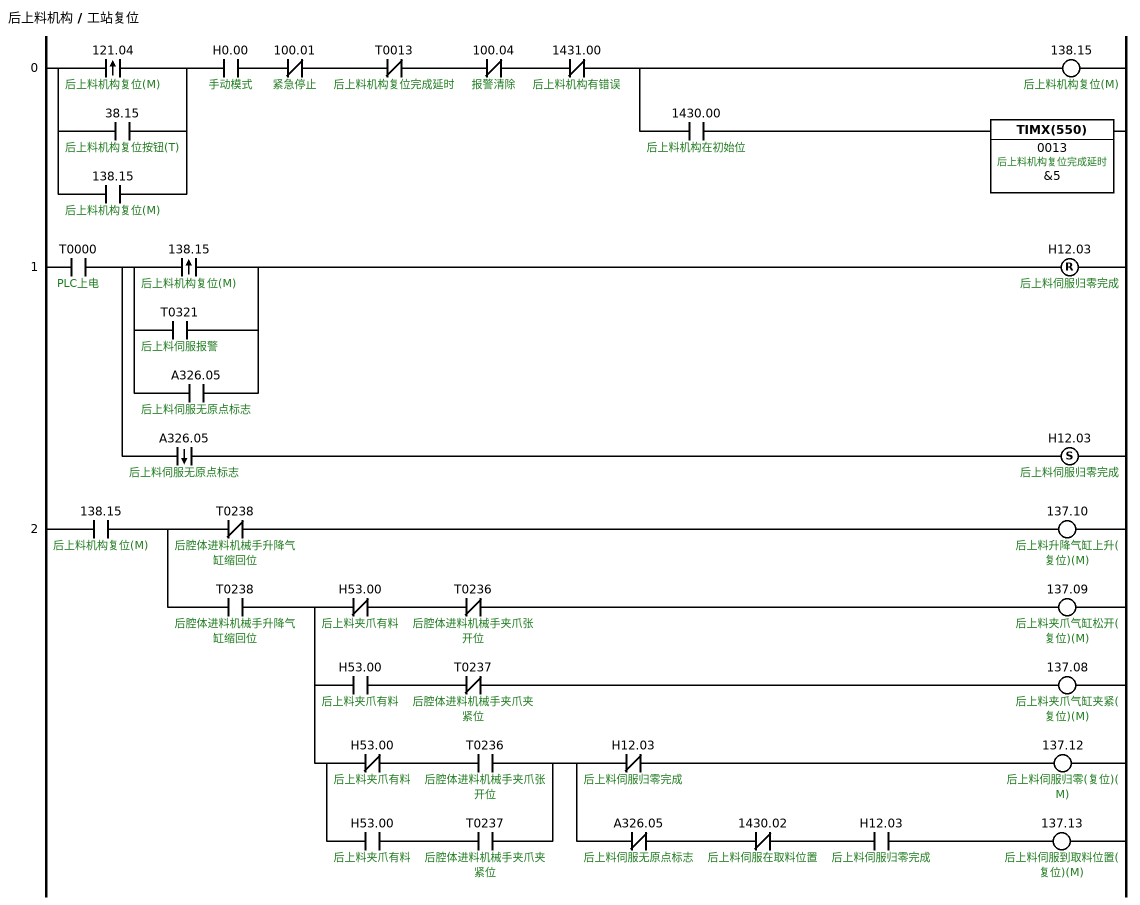
; rung 0
@LD 121.04  ; 后上料机构复位(M)
OR 38.15  ; 后上料机构复位按钮(T)
OR 138.15  ; 后上料机构复位(M)
AND H0.00  ; 手动模式
ANDNOT 100.01  ; 紧急停止
ANDNOT T0013  ; 后上料机构复位完成延时
ANDNOT 100.04  ; 报警清除
ANDNOT 1431.00  ; 后上料机构有错误
OUT 138.15  ; 后上料机构复位(M)
AND 1430.00  ; 后上料机构在初始位
TIMX(550) 0013 &5  ; 后上料机构复位完成延时
; rung 1
LD T0000  ; PLC上电
OUT TR0
@LD 138.15  ; 后上料机构复位(M)
OR T0321  ; 后上料伺服报警
OR A326.05  ; 后上料伺服无原点标志
ANDLD
RSET H12.03  ; 后上料伺服归零完成
LD TR0
%AND A326.05  ; 后上料伺服无原点标志
SET H12.03  ; 后上料伺服归零完成
; rung 2
LD 138.15  ; 后上料机构复位(M)
OUT TR0
ANDNOT T0238  ; 后腔体进料机械手升降气缸缩回位
OUT 137.10  ; 后上料升降气缸上升(复位)(M)
LD TR0
AND T0238  ; 后腔体进料机械手升降气缸缩回位
OUT TR0
ANDNOT H53.00  ; 后上料夹爪有料
ANDNOT T0236  ; 后腔体进料机械手夹爪张开位
OUT 137.09  ; 后上料夹爪气缸松开(复位)(M)
LD TR0
AND H53.00  ; 后上料夹爪有料
ANDNOT T0237  ; 后腔体进料机械手夹爪夹紧位
OUT 137.08  ; 后上料夹爪气缸夹紧(复位)(M)
LD TR0
LDNOT H53.00  ; 后上料夹爪有料
AND T0236  ; 后腔体进料机械手夹爪张开位
LD H53.00  ; 后上料夹爪有料
AND T0237  ; 后腔体进料机械手夹爪夹紧位
ORLD
ANDLD
OUT TR0
ANDNOT H12.03  ; 后上料伺服归零完成
OUT 137.12  ; 后上料伺服归零(复位)(M)
LD TR0
ANDNOT A326.05  ; 后上料伺服无原点标志
ANDNOT 1430.02  ; 后上料伺服在取料位置
AND H12.03  ; 后上料伺服归零完成
OUT 137.13  ; 后上料伺服到取料位置(复位)(M)

### Section 手动操作

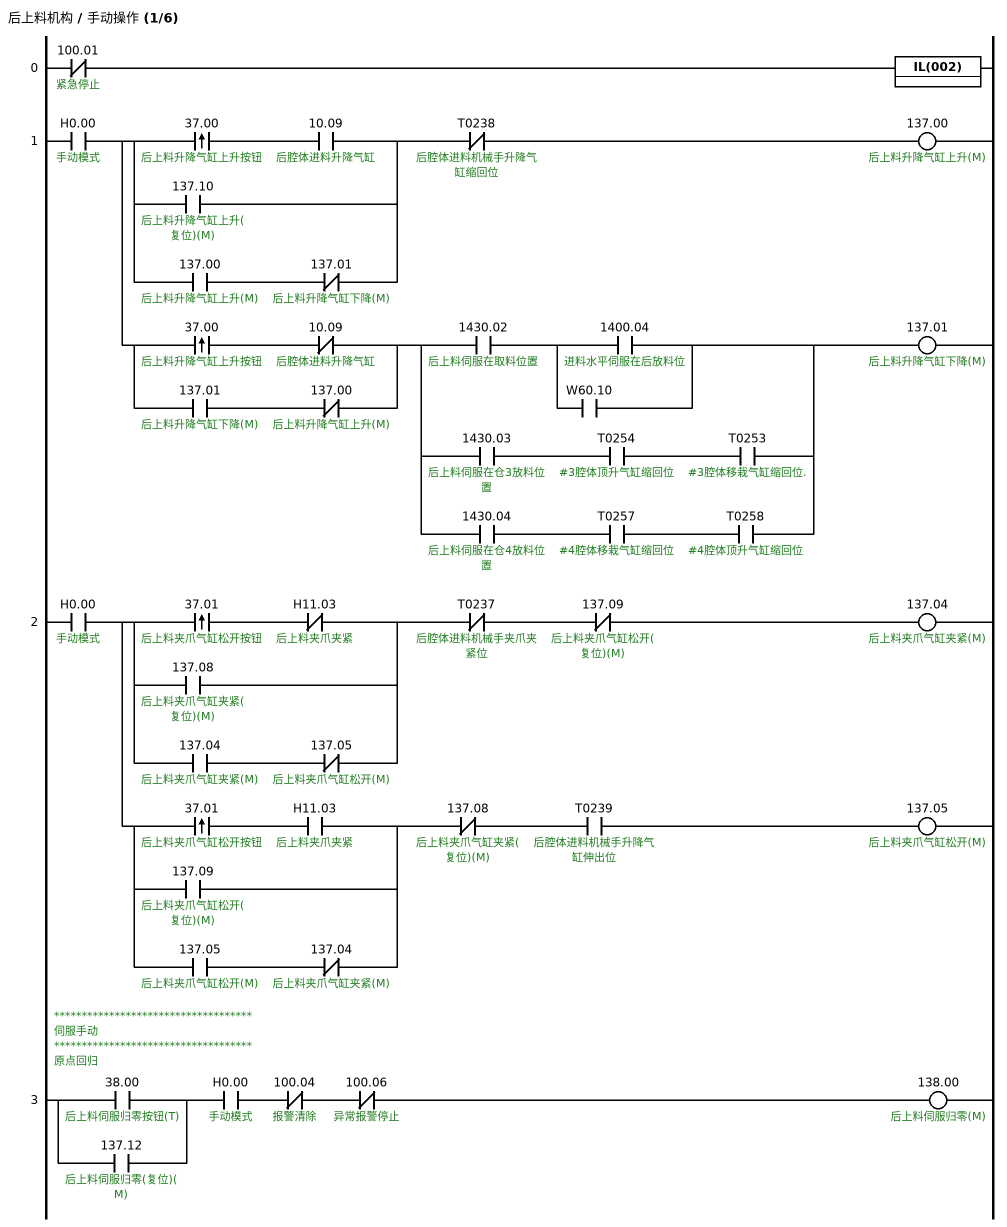
; rung 0
LDNOT 100.01  ; 紧急停止
IL(002)
; rung 1
LD H0.00  ; 手动模式
OUT TR0
@LD 37.00  ; 后上料升降气缸上升按钮
AND 10.09  ; 后腔体进料升降气缸
OR 137.10  ; 后上料升降气缸上升(复位)(M)
LD 137.00  ; 后上料升降气缸上升(M)
ANDNOT 137.01  ; 后上料升降气缸下降(M)
ORLD
ANDLD
ANDNOT T0238  ; 后腔体进料机械手升降气缸缩回位
OUT 137.00  ; 后上料升降气缸上升(M)
LD TR0
@LD 37.00  ; 后上料升降气缸上升按钮
ANDNOT 10.09  ; 后腔体进料升降气缸
LD 137.01  ; 后上料升降气缸下降(M)
ANDNOT 137.00  ; 后上料升降气缸上升(M)
ORLD
ANDLD
LD 1430.02  ; 后上料伺服在取料位置
LD 1400.04  ; 进料水平伺服在后放料位
OR W60.10
ANDLD
LD 1430.03  ; 后上料伺服在仓3放料位置
AND T0254  ; #3腔体顶升气缸缩回位
AND T0253  ; #3腔体移栽气缸缩回位.
ORLD
LD 1430.04  ; 后上料伺服在仓4放料位置
AND T0257  ; #4腔体移栽气缸缩回位
AND T0258  ; #4腔体顶升气缸缩回位
ORLD
ANDLD
OUT 137.01  ; 后上料升降气缸下降(M)
; rung 2
LD H0.00  ; 手动模式
OUT TR0
@LD 37.01  ; 后上料夹爪气缸松开按钮
ANDNOT H11.03  ; 后上料夹爪夹紧
OR 137.08  ; 后上料夹爪气缸夹紧(复位)(M)
LD 137.04  ; 后上料夹爪气缸夹紧(M)
ANDNOT 137.05  ; 后上料夹爪气缸松开(M)
ORLD
ANDLD
ANDNOT T0237  ; 后腔体进料机械手夹爪夹紧位
ANDNOT 137.09  ; 后上料夹爪气缸松开(复位)(M)
OUT 137.04  ; 后上料夹爪气缸夹紧(M)
LD TR0
@LD 37.01  ; 后上料夹爪气缸松开按钮
AND H11.03  ; 后上料夹爪夹紧
OR 137.09  ; 后上料夹爪气缸松开(复位)(M)
LD 137.05  ; 后上料夹爪气缸松开(M)
ANDNOT 137.04  ; 后上料夹爪气缸夹紧(M)
ORLD
ANDLD
ANDNOT 137.08  ; 后上料夹爪气缸夹紧(复位)(M)
AND T0239  ; 后腔体进料机械手升降气缸伸出位
OUT 137.05  ; 后上料夹爪气缸松开(M)
; rung 3: ************************************ / 伺服手动 / ************************************ / 原点回归
LD 38.00  ; 后上料伺服归零按钮(T)
OR 137.12  ; 后上料伺服归零(复位)(M)
AND H0.00  ; 手动模式
ANDNOT 100.04  ; 报警清除
ANDNOT 100.06  ; 异常报警停止
OUT 138.00  ; 后上料伺服归零(M)

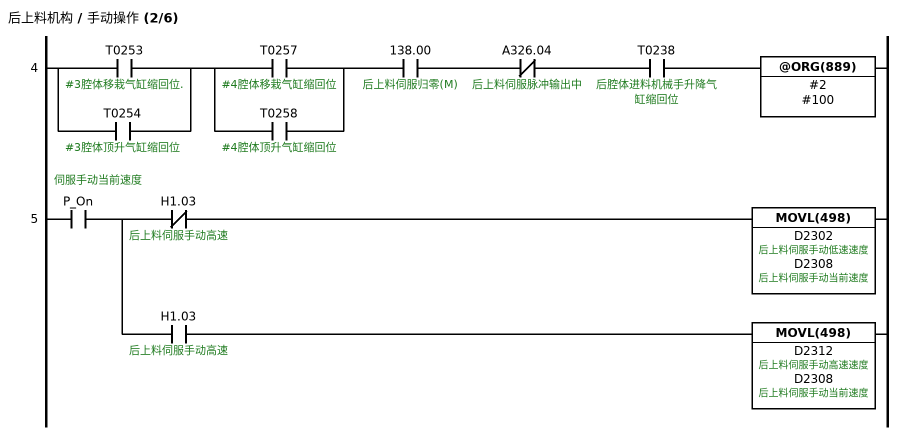
; rung 4
LD T0253  ; #3腔体移栽气缸缩回位.
OR T0254  ; #3腔体顶升气缸缩回位
LD T0257  ; #4腔体移栽气缸缩回位
OR T0258  ; #4腔体顶升气缸缩回位
ANDLD
AND 138.00  ; 后上料伺服归零(M)
ANDNOT A326.04  ; 后上料伺服脉冲输出中
AND T0238  ; 后腔体进料机械手升降气缸缩回位
@ORG(889) #2 #100
; rung 5: 伺服手动当前速度
LD P_On
OUT TR0
ANDNOT H1.03  ; 后上料伺服手动高速
MOVL(498) D2302 D2308  ; 后上料伺服手动低速速度, 后上料伺服手动当前速度
LD TR0
AND H1.03  ; 后上料伺服手动高速
MOVL(498) D2312 D2308  ; 后上料伺服手动高速速度, 后上料伺服手动当前速度

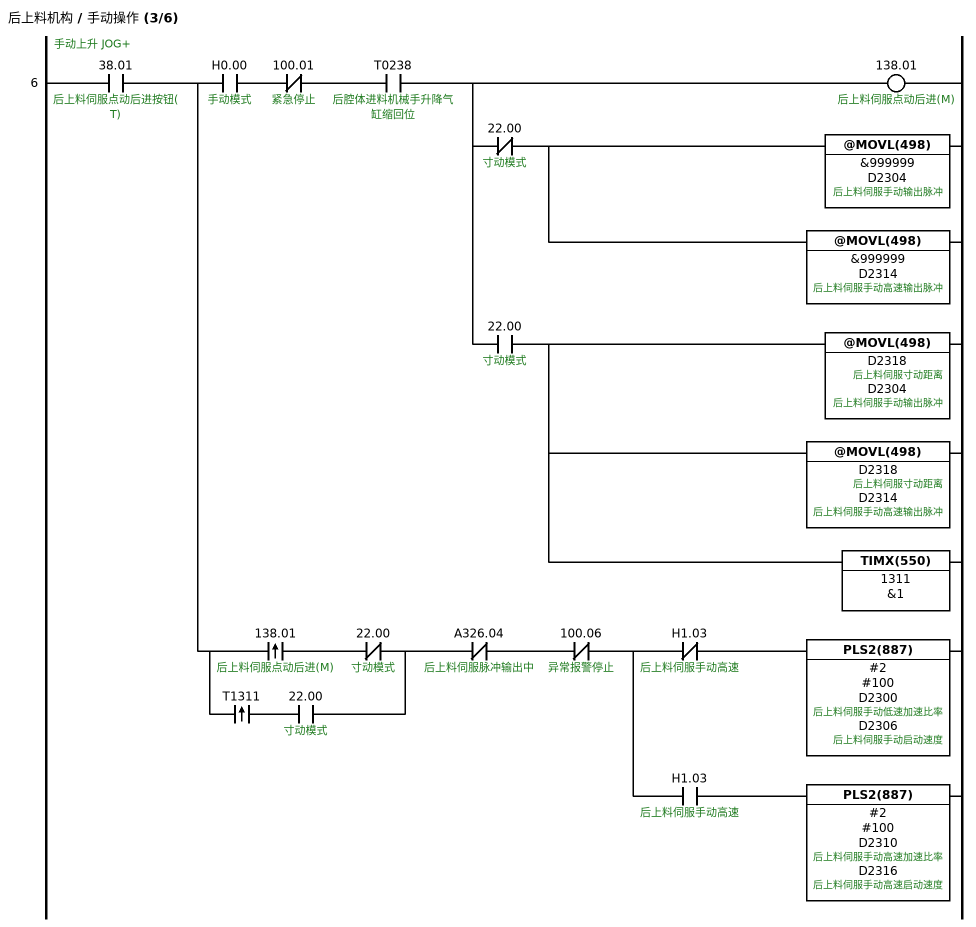
; rung 6: 手动上升 JOG+
LD 38.01  ; 后上料伺服点动后进按钮(T)
OUT TR0
AND H0.00  ; 手动模式
ANDNOT 100.01  ; 紧急停止
AND T0238  ; 后腔体进料机械手升降气缸缩回位
OUT TR1
OUT 138.01  ; 后上料伺服点动后进(M)
ANDNOT 22.00  ; 寸动模式
@MOVL(498) &999999 D2304  ; 后上料伺服手动输出脉冲
@MOVL(498) &999999 D2314  ; 后上料伺服手动高速输出脉冲
LD TR1
AND 22.00  ; 寸动模式
@MOVL(498) D2318 D2304  ; 后上料伺服寸动距离, 后上料伺服手动输出脉冲
@MOVL(498) D2318 D2314  ; 后上料伺服寸动距离, 后上料伺服手动高速输出脉冲
TIMX(550) 1311 &1
LD TR0
@LD 138.01  ; 后上料伺服点动后进(M)
ANDNOT 22.00  ; 寸动模式
@LD T1311
AND 22.00  ; 寸动模式
ORLD
ANDLD
ANDNOT A326.04  ; 后上料伺服脉冲输出中
ANDNOT 100.06  ; 异常报警停止
OUT TR0
ANDNOT H1.03  ; 后上料伺服手动高速
PLS2(887) #2 #100 D2300 D2306  ; 后上料伺服手动低速加速比率, 后上料伺服手动启动速度
LD TR0
AND H1.03  ; 后上料伺服手动高速
PLS2(887) #2 #100 D2310 D2316  ; 后上料伺服手动高速加速比率, 后上料伺服手动高速启动速度

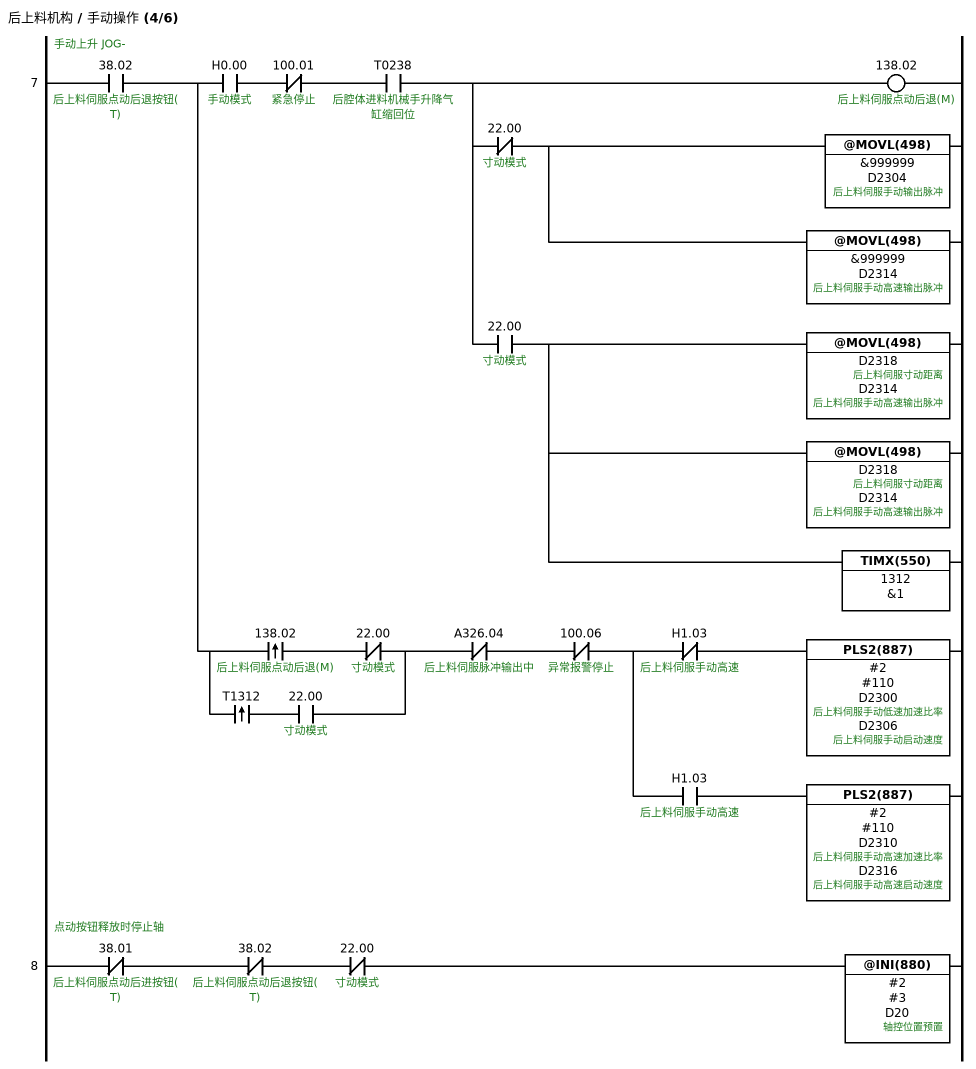
; rung 7: 手动上升 JOG-
LD 38.02  ; 后上料伺服点动后退按钮(T)
OUT TR0
AND H0.00  ; 手动模式
ANDNOT 100.01  ; 紧急停止
AND T0238  ; 后腔体进料机械手升降气缸缩回位
OUT TR1
OUT 138.02  ; 后上料伺服点动后退(M)
ANDNOT 22.00  ; 寸动模式
@MOVL(498) &999999 D2304  ; 后上料伺服手动输出脉冲
@MOVL(498) &999999 D2314  ; 后上料伺服手动高速输出脉冲
LD TR1
AND 22.00  ; 寸动模式
@MOVL(498) D2318 D2314  ; 后上料伺服寸动距离, 后上料伺服手动高速输出脉冲
@MOVL(498) D2318 D2314  ; 后上料伺服寸动距离, 后上料伺服手动高速输出脉冲
TIMX(550) 1312 &1
LD TR0
@LD 138.02  ; 后上料伺服点动后退(M)
ANDNOT 22.00  ; 寸动模式
@LD T1312
AND 22.00  ; 寸动模式
ORLD
ANDLD
ANDNOT A326.04  ; 后上料伺服脉冲输出中
ANDNOT 100.06  ; 异常报警停止
OUT TR0
ANDNOT H1.03  ; 后上料伺服手动高速
PLS2(887) #2 #110 D2300 D2306  ; 后上料伺服手动低速加速比率, 后上料伺服手动启动速度
LD TR0
AND H1.03  ; 后上料伺服手动高速
PLS2(887) #2 #110 D2310 D2316  ; 后上料伺服手动高速加速比率, 后上料伺服手动高速启动速度
; rung 8: 点动按钮释放时停止轴
LDNOT 38.01  ; 后上料伺服点动后进按钮(T)
ANDNOT 38.02  ; 后上料伺服点动后退按钮(T)
ANDNOT 22.00  ; 寸动模式
@INI(880) #2 #3 D20  ; 轴控位置预置

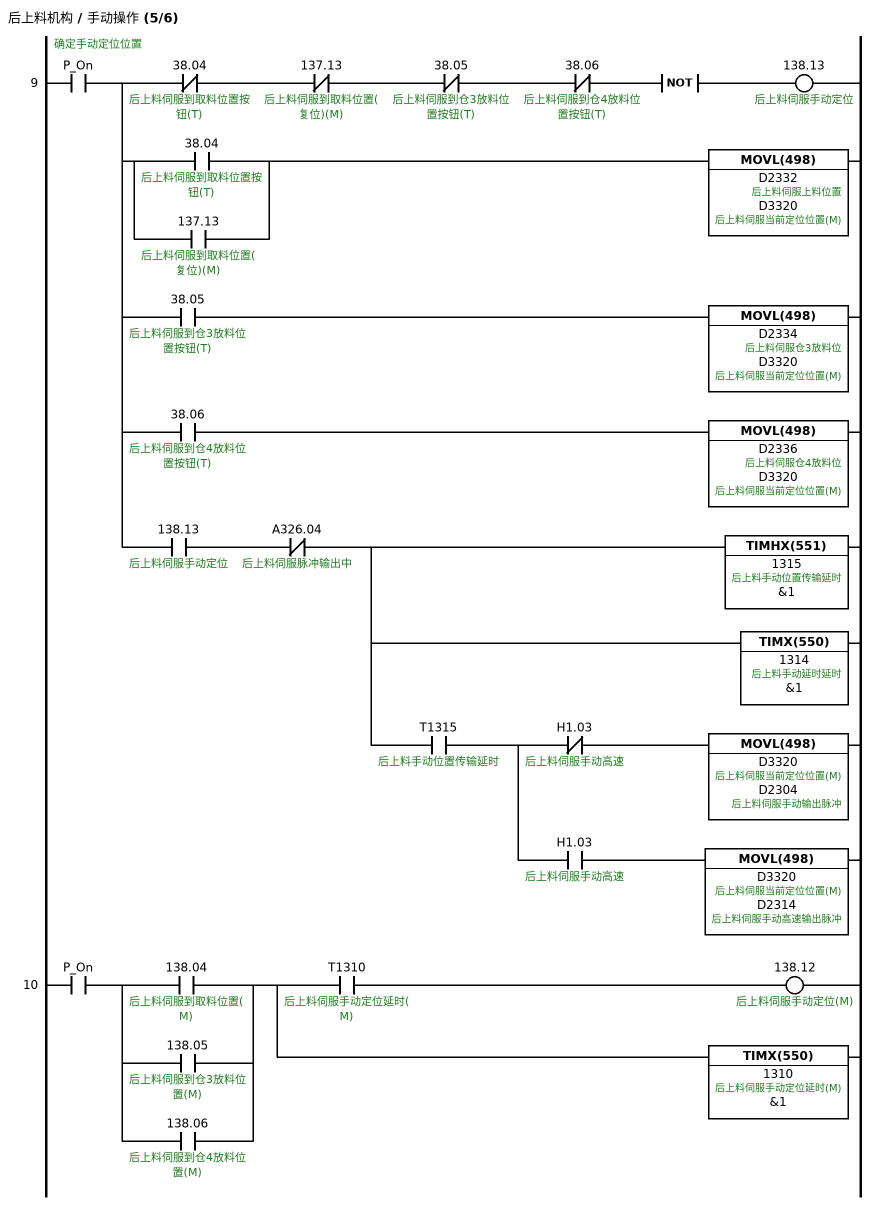
; rung 9: 确定手动定位位置
LD P_On
OUT TR0
ANDNOT 38.04  ; 后上料伺服到取料位置按钮(T)
ANDNOT 137.13  ; 后上料伺服到取料位置(复位)(M)
ANDNOT 38.05  ; 后上料伺服到仓3放料位置按钮(T)
ANDNOT 38.06  ; 后上料伺服到仓4放料位置按钮(T)
NOT(520)
OUT 138.13  ; 后上料伺服手动定位
LD TR0
LD 38.04  ; 后上料伺服到取料位置按钮(T)
OR 137.13  ; 后上料伺服到取料位置(复位)(M)
ANDLD
MOVL(498) D2332 D3320  ; 后上料伺服上料位置, 后上料伺服当前定位位置(M)
LD TR0
AND 38.05  ; 后上料伺服到仓3放料位置按钮(T)
MOVL(498) D2334 D3320  ; 后上料伺服仓3放料位, 后上料伺服当前定位位置(M)
LD TR0
AND 38.06  ; 后上料伺服到仓4放料位置按钮(T)
MOVL(498) D2336 D3320  ; 后上料伺服仓4放料位, 后上料伺服当前定位位置(M)
LD TR0
AND 138.13  ; 后上料伺服手动定位
ANDNOT A326.04  ; 后上料伺服脉冲输出中
TIMHX(551) 1315 &1  ; 后上料手动位置传输延时
TIMX(550) 1314 &1  ; 后上料手动延时延时
AND T1315  ; 后上料手动位置传输延时
OUT TR0
ANDNOT H1.03  ; 后上料伺服手动高速
MOVL(498) D3320 D2304  ; 后上料伺服当前定位位置(M), 后上料伺服手动输出脉冲
LD TR0
AND H1.03  ; 后上料伺服手动高速
MOVL(498) D3320 D2314  ; 后上料伺服当前定位位置(M), 后上料伺服手动高速输出脉冲
; rung 10
LD P_On
LD 138.04  ; 后上料伺服到取料位置(M)
OR 138.05  ; 后上料伺服到仓3放料位置(M)
OR 138.06  ; 后上料伺服到仓4放料位置(M)
ANDLD
OUT TR0
AND T1310  ; 后上料伺服手动定位延时(M)
OUT 138.12  ; 后上料伺服手动定位(M)
LD TR0
TIMX(550) 1310 &1  ; 后上料伺服手动定位延时(M)

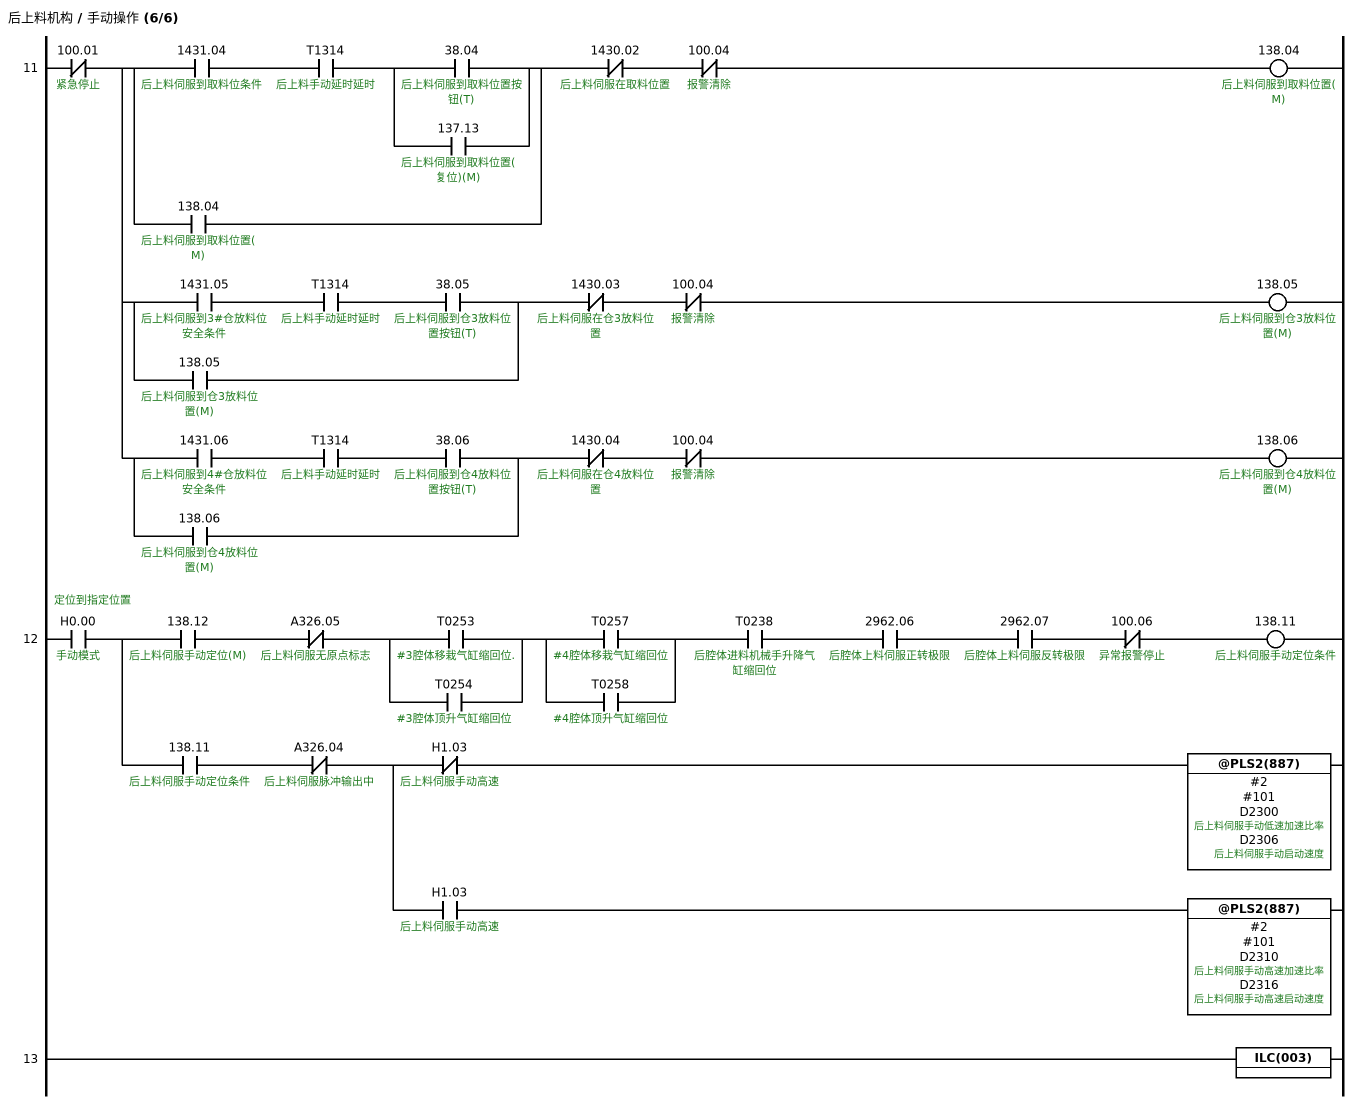
; rung 11
LDNOT 100.01  ; 紧急停止
OUT TR0
LD 1431.04  ; 后上料伺服到取料位条件
AND T1314  ; 后上料手动延时延时
LD 38.04  ; 后上料伺服到取料位置按钮(T)
OR 137.13  ; 后上料伺服到取料位置(复位)(M)
ANDLD
OR 138.04  ; 后上料伺服到取料位置(M)
ANDLD
ANDNOT 1430.02  ; 后上料伺服在取料位置
ANDNOT 100.04  ; 报警清除
OUT 138.04  ; 后上料伺服到取料位置(M)
LD TR0
LD 1431.05  ; 后上料伺服到3#仓放料位安全条件
AND T1314  ; 后上料手动延时延时
AND 38.05  ; 后上料伺服到仓3放料位置按钮(T)
OR 138.05  ; 后上料伺服到仓3放料位置(M)
ANDLD
ANDNOT 1430.03  ; 后上料伺服在仓3放料位置
ANDNOT 100.04  ; 报警清除
OUT 138.05  ; 后上料伺服到仓3放料位置(M)
LD TR0
LD 1431.06  ; 后上料伺服到4#仓放料位安全条件
AND T1314  ; 后上料手动延时延时
AND 38.06  ; 后上料伺服到仓4放料位置按钮(T)
OR 138.06  ; 后上料伺服到仓4放料位置(M)
ANDLD
ANDNOT 1430.04  ; 后上料伺服在仓4放料位置
ANDNOT 100.04  ; 报警清除
OUT 138.06  ; 后上料伺服到仓4放料位置(M)
; rung 12: 定位到指定位置
LD H0.00  ; 手动模式
OUT TR0
AND 138.12  ; 后上料伺服手动定位(M)
ANDNOT A326.05  ; 后上料伺服无原点标志
LD T0253  ; #3腔体移栽气缸缩回位.
OR T0254  ; #3腔体顶升气缸缩回位
ANDLD
LD T0257  ; #4腔体移栽气缸缩回位
OR T0258  ; #4腔体顶升气缸缩回位
ANDLD
AND T0238  ; 后腔体进料机械手升降气缸缩回位
AND 2962.06  ; 后腔体上料伺服正转极限
AND 2962.07  ; 后腔体上料伺服反转极限
ANDNOT 100.06  ; 异常报警停止
OUT 138.11  ; 后上料伺服手动定位条件
LD TR0
AND 138.11  ; 后上料伺服手动定位条件
ANDNOT A326.04  ; 后上料伺服脉冲输出中
OUT TR0
ANDNOT H1.03  ; 后上料伺服手动高速
@PLS2(887) #2 #101 D2300 D2306  ; 后上料伺服手动低速加速比率, 后上料伺服手动启动速度
LD TR0
AND H1.03  ; 后上料伺服手动高速
@PLS2(887) #2 #101 D2310 D2316  ; 后上料伺服手动高速加速比率, 后上料伺服手动高速启动速度
; rung 13
ILC(003)

### Section 自动运行

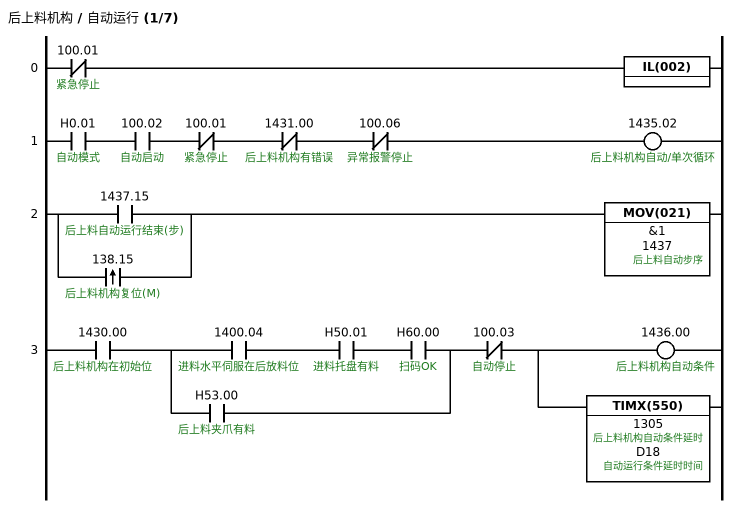
; rung 0
LDNOT 100.01  ; 紧急停止
IL(002)
; rung 1
LD H0.01  ; 自动模式
AND 100.02  ; 自动启动
ANDNOT 100.01  ; 紧急停止
ANDNOT 1431.00  ; 后上料机构有错误
ANDNOT 100.06  ; 异常报警停止
OUT 1435.02  ; 后上料机构自动/单次循环
; rung 2
LD 1437.15  ; 后上料自动运行结束(步)
@OR 138.15  ; 后上料机构复位(M)
MOV(021) &1 1437  ; 后上料自动步序
; rung 3
LD 1430.00  ; 后上料机构在初始位
LD 1400.04  ; 进料水平伺服在后放料位
AND H50.01  ; 进料托盘有料
AND H60.00  ; 扫码OK
OR H53.00  ; 后上料夹爪有料
ANDLD
ANDNOT 100.03  ; 自动停止
OUT 1436.00  ; 后上料机构自动条件
TIMX(550) 1305 D18  ; 自动运行条件延时时间, 后上料机构自动条件延时

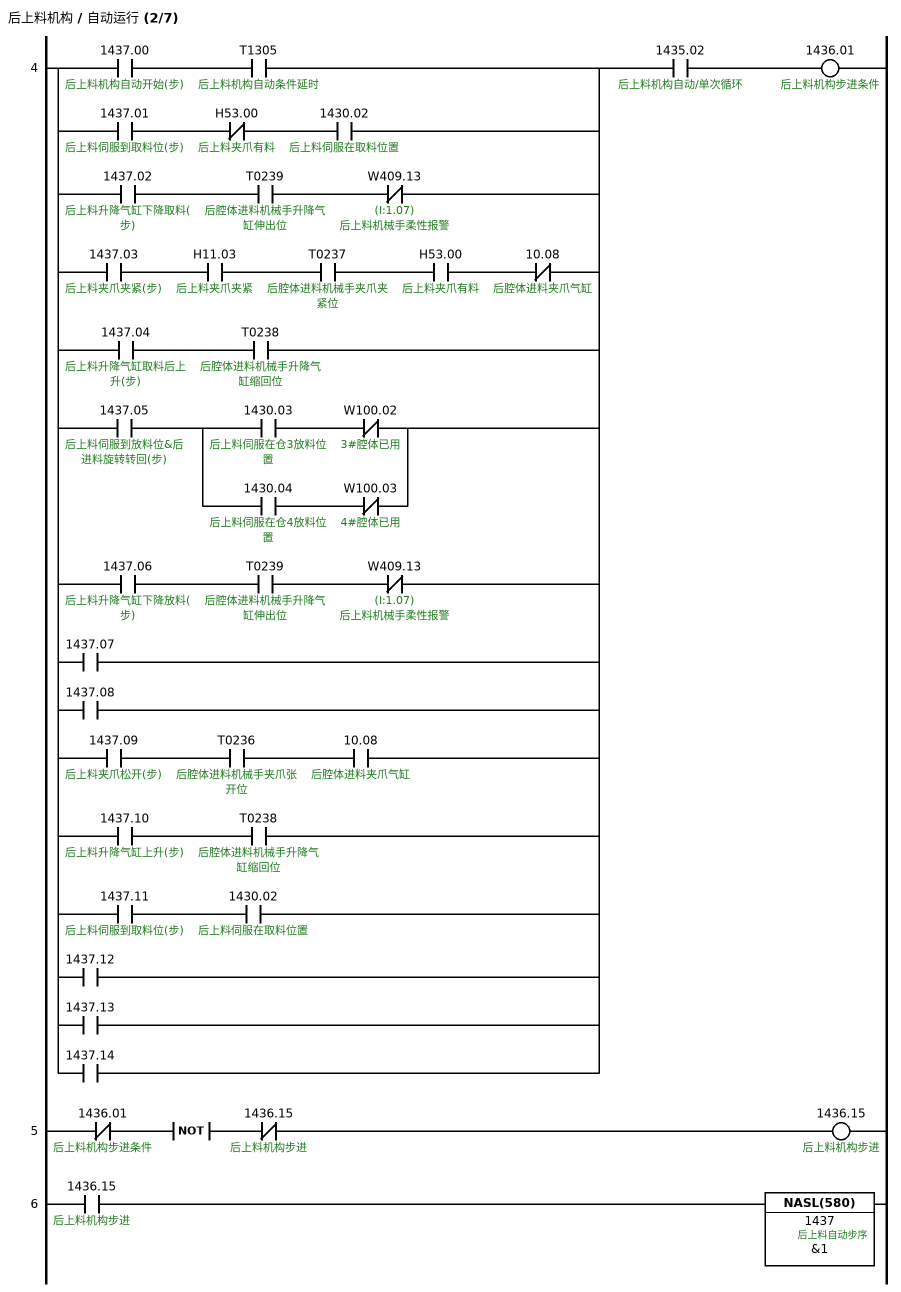
; rung 4
LD 1437.00  ; 后上料机构自动开始(步)
AND T1305  ; 后上料机构自动条件延时
LD 1437.01  ; 后上料伺服到取料位(步)
ANDNOT H53.00  ; 后上料夹爪有料
AND 1430.02  ; 后上料伺服在取料位置
ORLD
LD 1437.02  ; 后上料升降气缸下降取料(步)
AND T0239  ; 后腔体进料机械手升降气缸伸出位
ANDNOT W409.13  ; (I:1.07) 后上料机械手柔性报警
ORLD
LD 1437.03  ; 后上料夹爪夹紧(步)
AND H11.03  ; 后上料夹爪夹紧
AND T0237  ; 后腔体进料机械手夹爪夹紧位
AND H53.00  ; 后上料夹爪有料
ANDNOT 10.08  ; 后腔体进料夹爪气缸
ORLD
LD 1437.04  ; 后上料升降气缸取料后上升(步)
AND T0238  ; 后腔体进料机械手升降气缸缩回位
ORLD
LD 1437.05  ; 后上料伺服到放料位&后进料旋转转回(步)
LD 1430.03  ; 后上料伺服在仓3放料位置
ANDNOT W100.02  ; 3#腔体已用
LD 1430.04  ; 后上料伺服在仓4放料位置
ANDNOT W100.03  ; 4#腔体已用
ORLD
ANDLD
ORLD
LD 1437.06  ; 后上料升降气缸下降放料(步)
AND T0239  ; 后腔体进料机械手升降气缸伸出位
ANDNOT W409.13  ; (I:1.07) 后上料机械手柔性报警
ORLD
OR 1437.07
OR 1437.08
LD 1437.09  ; 后上料夹爪松开(步)
AND T0236  ; 后腔体进料机械手夹爪张开位
AND 10.08  ; 后腔体进料夹爪气缸
ORLD
LD 1437.10  ; 后上料升降气缸上升(步)
AND T0238  ; 后腔体进料机械手升降气缸缩回位
ORLD
LD 1437.11  ; 后上料伺服到取料位(步)
AND 1430.02  ; 后上料伺服在取料位置
ORLD
OR 1437.12
OR 1437.13
OR 1437.14
AND 1435.02  ; 后上料机构自动/单次循环
OUT 1436.01  ; 后上料机构步进条件
; rung 5
LDNOT 1436.01  ; 后上料机构步进条件
NOT(520)
ANDNOT 1436.15  ; 后上料机构步进
OUT 1436.15  ; 后上料机构步进
; rung 6
LD 1436.15  ; 后上料机构步进
NASL(580) 1437 &1  ; 后上料自动步序

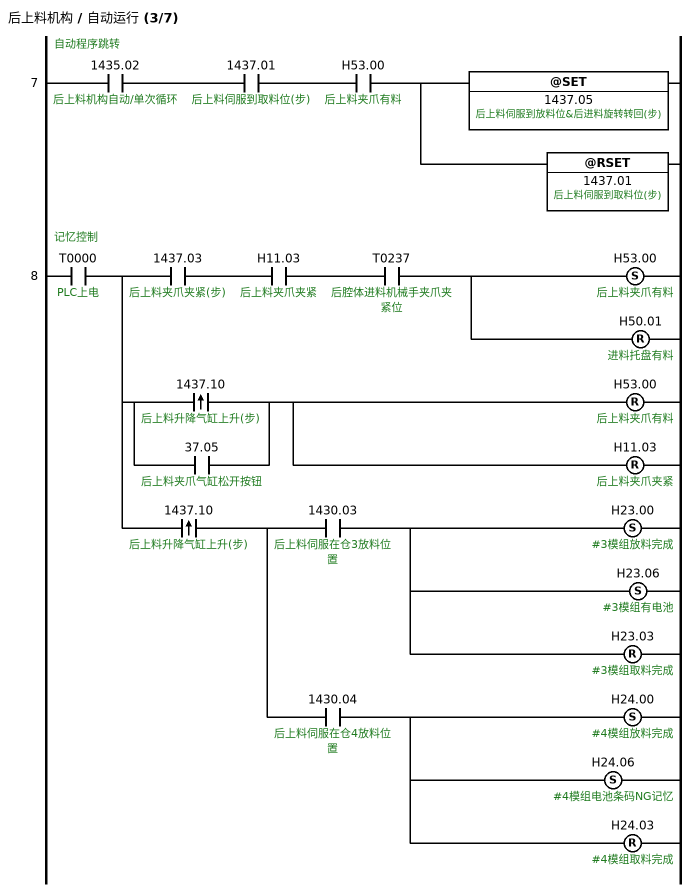
; rung 7: 自动程序跳转
LD 1435.02  ; 后上料机构自动/单次循环
AND 1437.01  ; 后上料伺服到取料位(步)
AND H53.00  ; 后上料夹爪有料
@SET 1437.05  ; 后上料伺服到放料位&后进料旋转转回(步)
@RSET 1437.01  ; 后上料伺服到取料位(步)
; rung 8: 记忆控制
LD T0000  ; PLC上电
OUT TR0
AND 1437.03  ; 后上料夹爪夹紧(步)
AND H11.03  ; 后上料夹爪夹紧
AND T0237  ; 后腔体进料机械手夹爪夹紧位
SET H53.00  ; 后上料夹爪有料
RSET H50.01  ; 进料托盘有料
LD TR0
@LD 1437.10  ; 后上料升降气缸上升(步)
OR 37.05  ; 后上料夹爪气缸松开按钮
ANDLD
RSET H53.00  ; 后上料夹爪有料
RSET H11.03  ; 后上料夹爪夹紧
LD TR0
@AND 1437.10  ; 后上料升降气缸上升(步)
OUT TR0
AND 1430.03  ; 后上料伺服在仓3放料位置
SET H23.00  ; #3模组放料完成
SET H23.06  ; #3模组有电池
RSET H23.03  ; #3模组取料完成
LD TR0
AND 1430.04  ; 后上料伺服在仓4放料位置
SET H24.00  ; #4模组放料完成
SET H24.06  ; #4模组电池条码NG记忆
RSET H24.03  ; #4模组取料完成

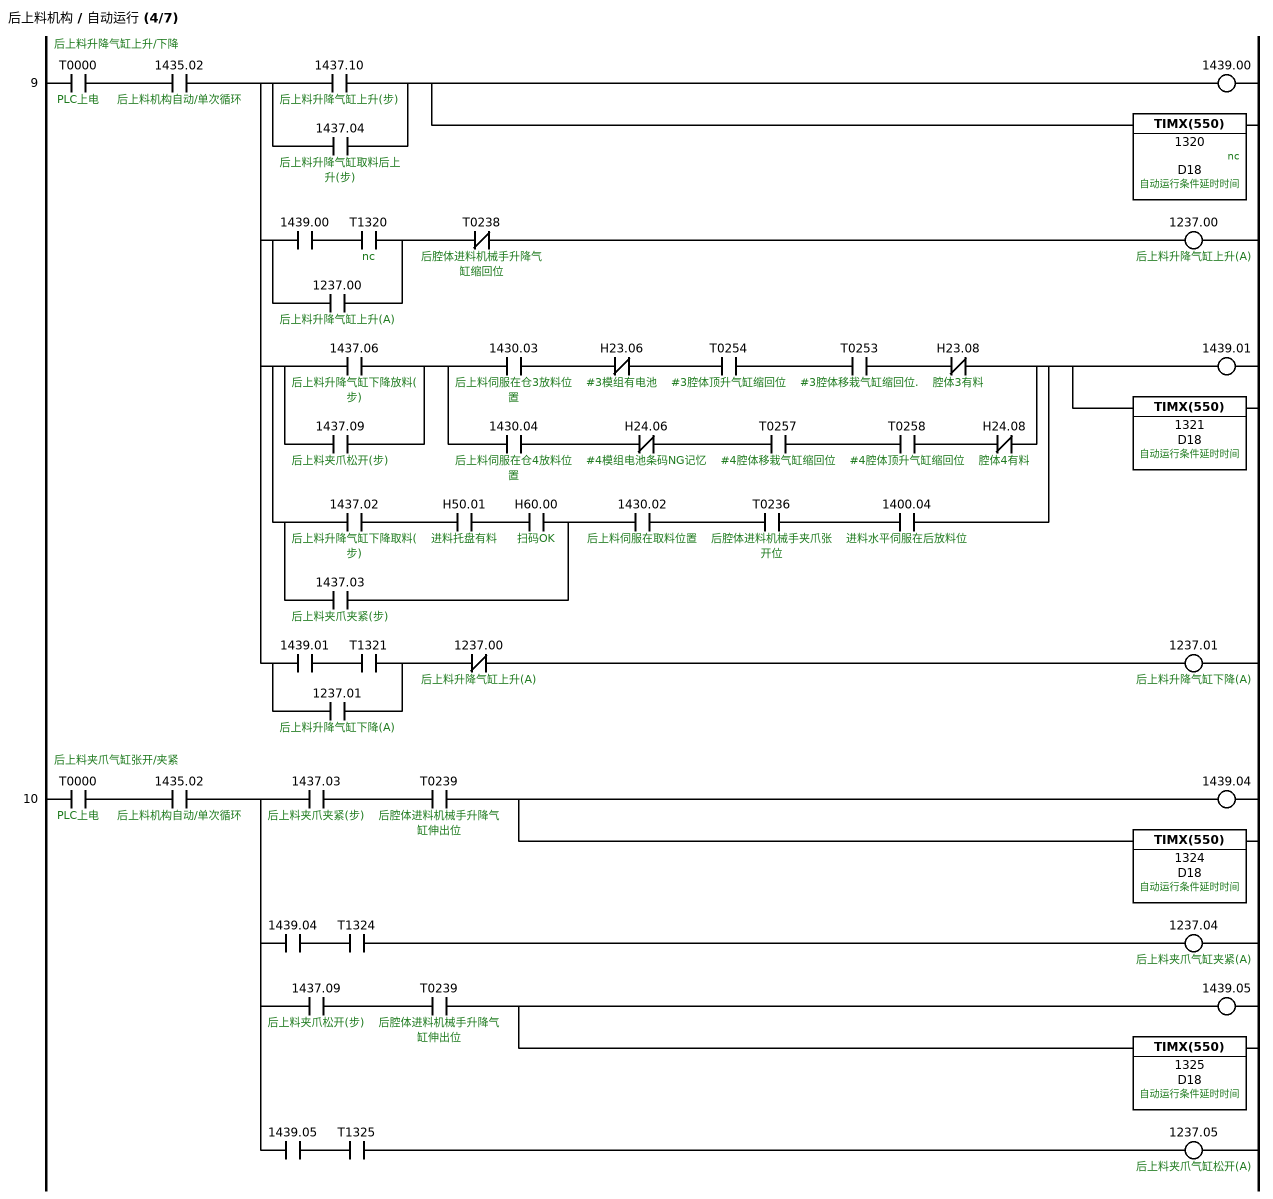
; rung 9: 后上料升降气缸上升/下降
LD T0000  ; PLC上电
AND 1435.02  ; 后上料机构自动/单次循环
OUT TR0
LD 1437.10  ; 后上料升降气缸上升(步)
OR 1437.04  ; 后上料升降气缸取料后上升(步)
ANDLD
OUT 1439.00
TIMX(550) 1320 D18  ; 自动运行条件延时时间, nc
LD TR0
LD 1439.00
AND T1320  ; nc
OR 1237.00  ; 后上料升降气缸上升(A)
ANDLD
ANDNOT T0238  ; 后腔体进料机械手升降气缸缩回位
OUT 1237.00  ; 后上料升降气缸上升(A)
LD TR0
LD 1437.06  ; 后上料升降气缸下降放料(步)
OR 1437.09  ; 后上料夹爪松开(步)
LD 1430.03  ; 后上料伺服在仓3放料位置
ANDNOT H23.06  ; #3模组有电池
AND T0254  ; #3腔体顶升气缸缩回位
AND T0253  ; #3腔体移栽气缸缩回位.
ANDNOT H23.08  ; 腔体3有料
LD 1430.04  ; 后上料伺服在仓4放料位置
ANDNOT H24.06  ; #4模组电池条码NG记忆
AND T0257  ; #4腔体移栽气缸缩回位
AND T0258  ; #4腔体顶升气缸缩回位
ANDNOT H24.08  ; 腔体4有料
ORLD
ANDLD
LD 1437.02  ; 后上料升降气缸下降取料(步)
AND H50.01  ; 进料托盘有料
AND H60.00  ; 扫码OK
OR 1437.03  ; 后上料夹爪夹紧(步)
AND 1430.02  ; 后上料伺服在取料位置
AND T0236  ; 后腔体进料机械手夹爪张开位
AND 1400.04  ; 进料水平伺服在后放料位
ORLD
ANDLD
OUT 1439.01
TIMX(550) 1321 D18  ; 自动运行条件延时时间
LD TR0
LD 1439.01
AND T1321
OR 1237.01  ; 后上料升降气缸下降(A)
ANDLD
ANDNOT 1237.00  ; 后上料升降气缸上升(A)
OUT 1237.01  ; 后上料升降气缸下降(A)
; rung 10: 后上料夹爪气缸张开/夹紧
LD T0000  ; PLC上电
AND 1435.02  ; 后上料机构自动/单次循环
OUT TR0
AND 1437.03  ; 后上料夹爪夹紧(步)
AND T0239  ; 后腔体进料机械手升降气缸伸出位
OUT 1439.04
TIMX(550) 1324 D18  ; 自动运行条件延时时间
LD TR0
AND 1439.04
AND T1324
OUT 1237.04  ; 后上料夹爪气缸夹紧(A)
LD TR0
AND 1437.09  ; 后上料夹爪松开(步)
AND T0239  ; 后腔体进料机械手升降气缸伸出位
OUT 1439.05
TIMX(550) 1325 D18  ; 自动运行条件延时时间
LD TR0
AND 1439.05
AND T1325
OUT 1237.05  ; 后上料夹爪气缸松开(A)

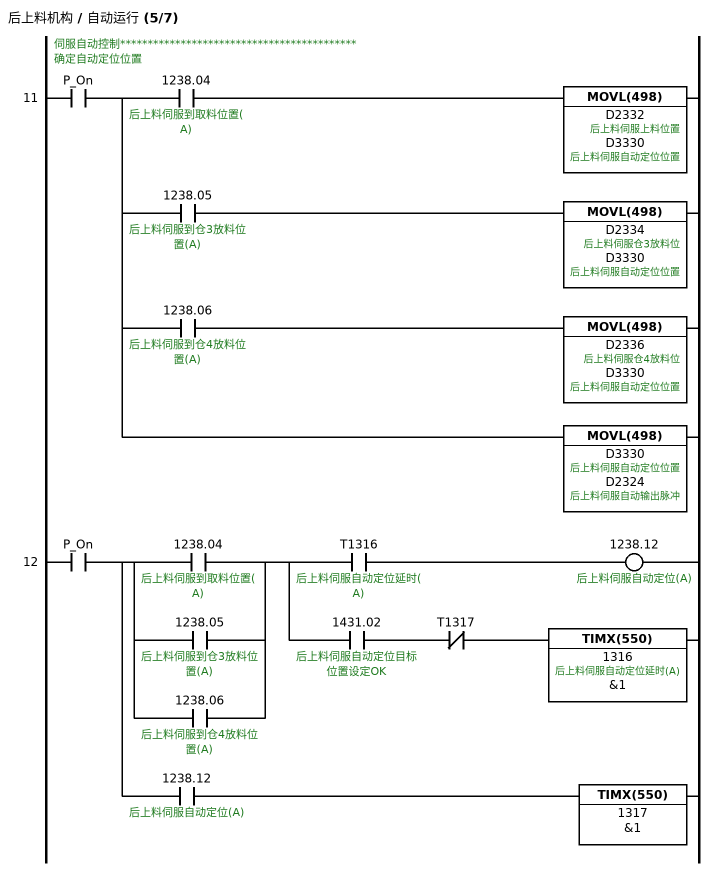
; rung 11: 伺服自动控制******************************************* / 确定自动定位位置
LD P_On
OUT TR0
AND 1238.04  ; 后上料伺服到取料位置(A)
MOVL(498) D2332 D3330  ; 后上料伺服上料位置, 后上料伺服自动定位位置
LD TR0
AND 1238.05  ; 后上料伺服到仓3放料位置(A)
MOVL(498) D2334 D3330  ; 后上料伺服仓3放料位, 后上料伺服自动定位位置
LD TR0
AND 1238.06  ; 后上料伺服到仓4放料位置(A)
MOVL(498) D2336 D3330  ; 后上料伺服仓4放料位, 后上料伺服自动定位位置
LD TR0
MOVL(498) D3330 D2324  ; 后上料伺服自动定位位置, 后上料伺服自动输出脉冲
; rung 12
LD P_On
OUT TR0
LD 1238.04  ; 后上料伺服到取料位置(A)
OR 1238.05  ; 后上料伺服到仓3放料位置(A)
OR 1238.06  ; 后上料伺服到仓4放料位置(A)
ANDLD
OUT TR1
AND T1316  ; 后上料伺服自动定位延时(A)
OUT 1238.12  ; 后上料伺服自动定位(A)
LD TR1
AND 1431.02  ; 后上料伺服自动定位目标位置设定OK
ANDNOT T1317
TIMX(550) 1316 &1  ; 后上料伺服自动定位延时(A)
LD TR0
AND 1238.12  ; 后上料伺服自动定位(A)
TIMX(550) 1317 &1

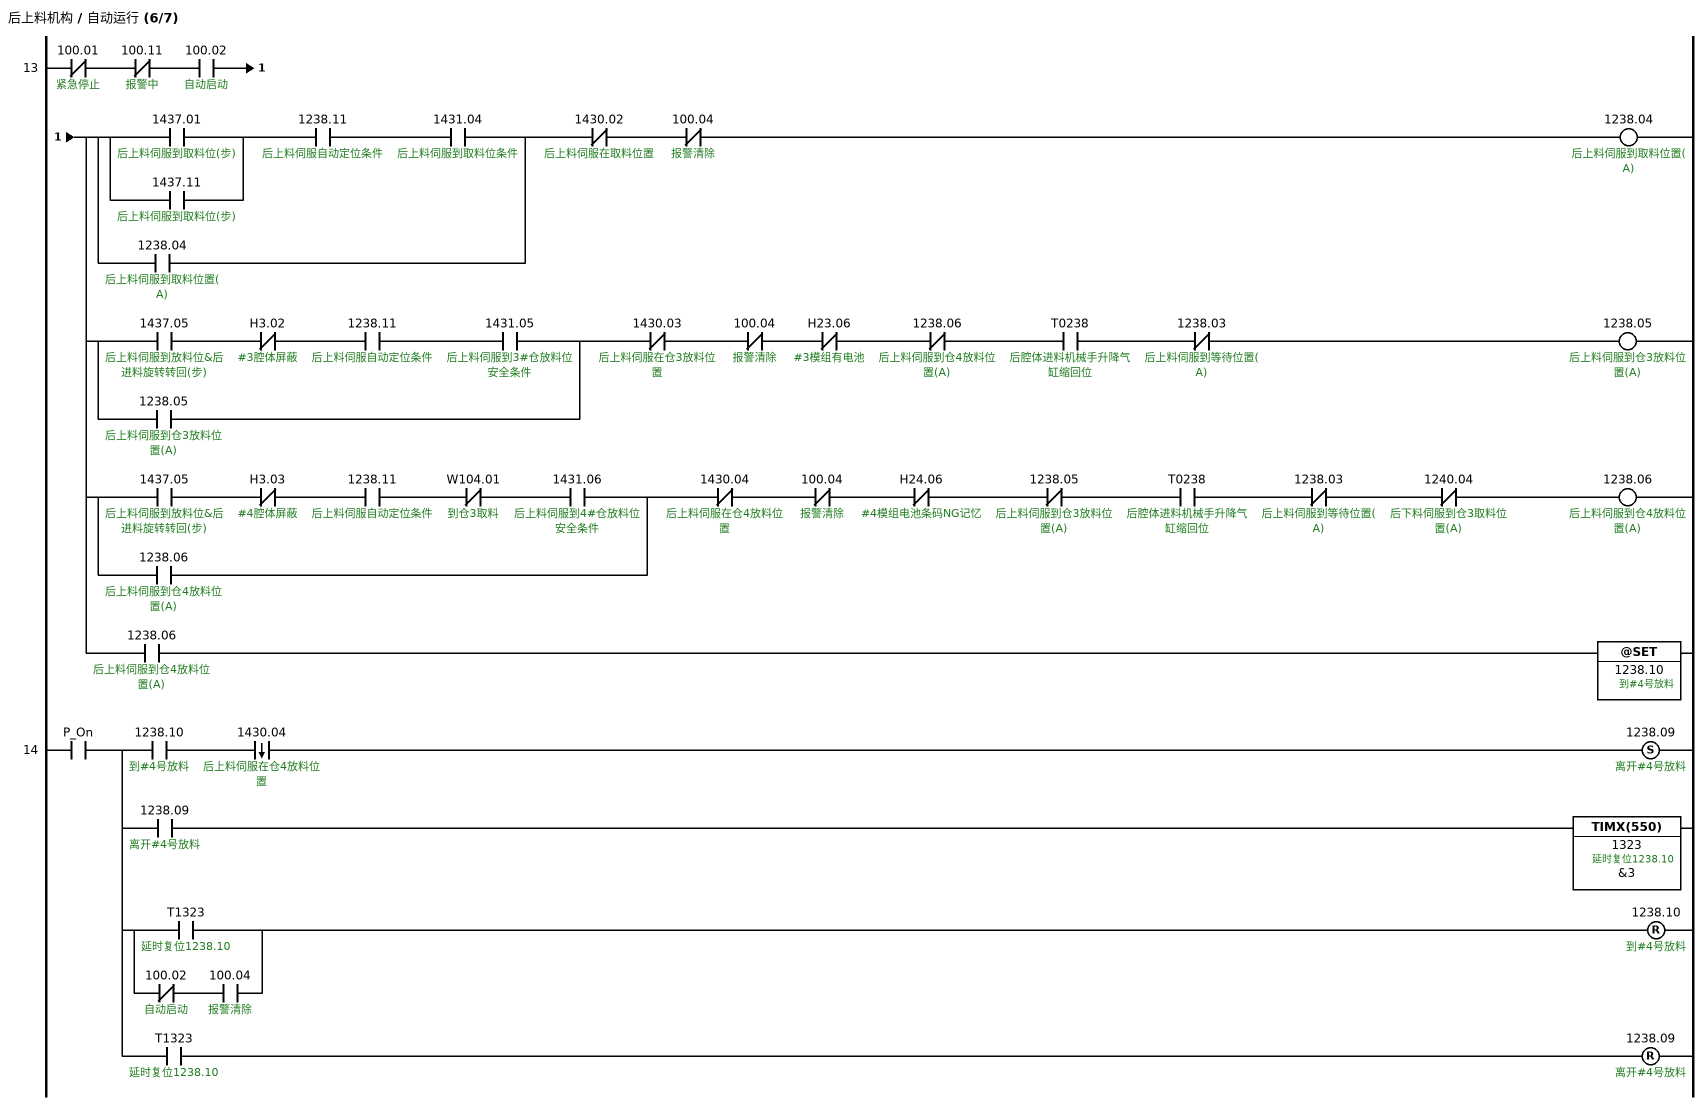
; rung 13
LDNOT 100.01  ; 紧急停止
ANDNOT 100.11  ; 报警中
AND 100.02  ; 自动启动
OUT TR0
LD 1437.01  ; 后上料伺服到取料位(步)
OR 1437.11  ; 后上料伺服到取料位(步)
AND 1238.11  ; 后上料伺服自动定位条件
AND 1431.04  ; 后上料伺服到取料位条件
OR 1238.04  ; 后上料伺服到取料位置(A)
ANDLD
ANDNOT 1430.02  ; 后上料伺服在取料位置
ANDNOT 100.04  ; 报警清除
OUT 1238.04  ; 后上料伺服到取料位置(A)
LD TR0
LD 1437.05  ; 后上料伺服到放料位&后进料旋转转回(步)
ANDNOT H3.02  ; #3腔体屏蔽
AND 1238.11  ; 后上料伺服自动定位条件
AND 1431.05  ; 后上料伺服到3#仓放料位安全条件
OR 1238.05  ; 后上料伺服到仓3放料位置(A)
ANDLD
ANDNOT 1430.03  ; 后上料伺服在仓3放料位置
ANDNOT 100.04  ; 报警清除
ANDNOT H23.06  ; #3模组有电池
ANDNOT 1238.06  ; 后上料伺服到仓4放料位置(A)
AND T0238  ; 后腔体进料机械手升降气缸缩回位
ANDNOT 1238.03  ; 后上料伺服到等待位置(A)
OUT 1238.05  ; 后上料伺服到仓3放料位置(A)
LD TR0
LD 1437.05  ; 后上料伺服到放料位&后进料旋转转回(步)
ANDNOT H3.03  ; #4腔体屏蔽
AND 1238.11  ; 后上料伺服自动定位条件
ANDNOT W104.01  ; 到仓3取料
AND 1431.06  ; 后上料伺服到4#仓放料位安全条件
OR 1238.06  ; 后上料伺服到仓4放料位置(A)
ANDLD
ANDNOT 1430.04  ; 后上料伺服在仓4放料位置
ANDNOT 100.04  ; 报警清除
ANDNOT H24.06  ; #4模组电池条码NG记忆
ANDNOT 1238.05  ; 后上料伺服到仓3放料位置(A)
AND T0238  ; 后腔体进料机械手升降气缸缩回位
ANDNOT 1238.03  ; 后上料伺服到等待位置(A)
ANDNOT 1240.04  ; 后下料伺服到仓3取料位置(A)
OUT 1238.06  ; 后上料伺服到仓4放料位置(A)
LD TR0
AND 1238.06  ; 后上料伺服到仓4放料位置(A)
@SET 1238.10  ; 到#4号放料
; rung 14
LD P_On
OUT TR0
AND 1238.10  ; 到#4号放料
%AND 1430.04  ; 后上料伺服在仓4放料位置
SET 1238.09  ; 离开#4号放料
LD TR0
AND 1238.09  ; 离开#4号放料
TIMX(550) 1323 &3  ; 延时复位1238.10
LD TR0
LD T1323  ; 延时复位1238.10
LDNOT 100.02  ; 自动启动
AND 100.04  ; 报警清除
ORLD
ANDLD
RSET 1238.10  ; 到#4号放料
LD TR0
AND T1323  ; 延时复位1238.10
RSET 1238.09  ; 离开#4号放料

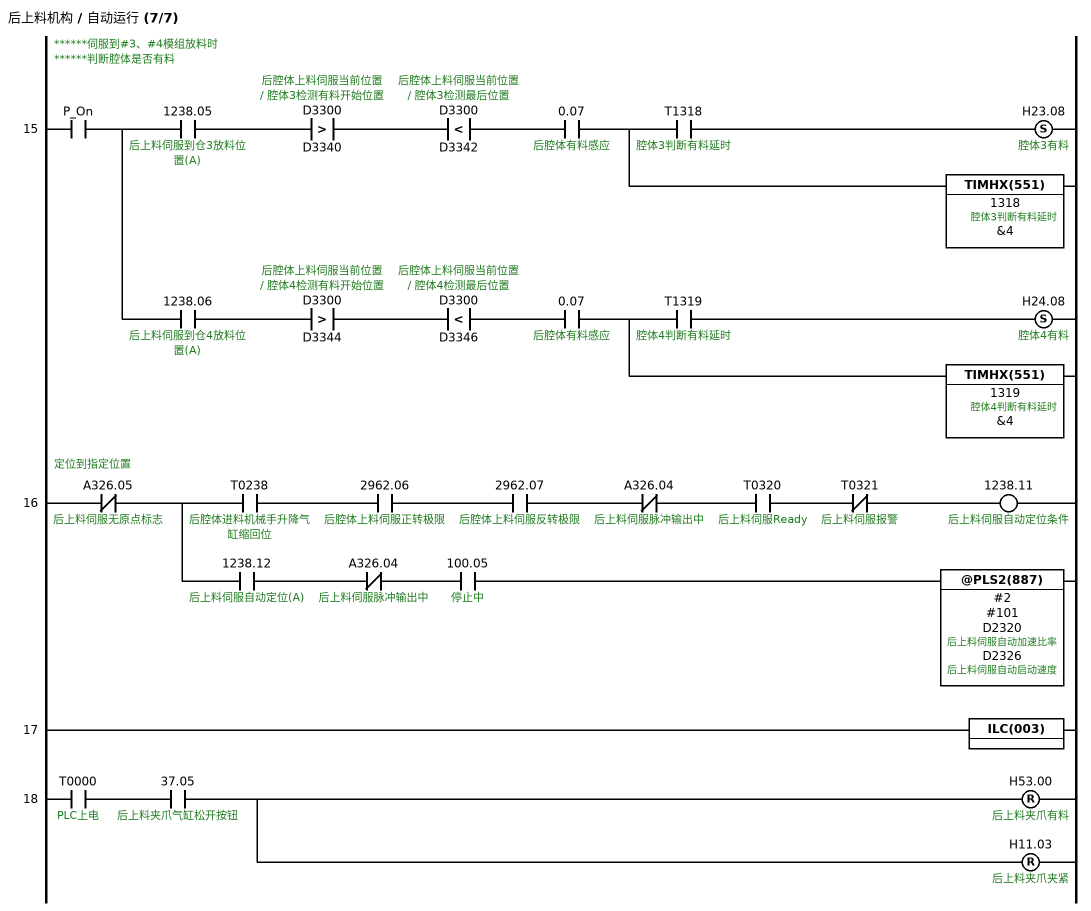
; rung 15: ******伺服到#3、#4模组放料时 / ******判断腔体是否有料
LD P_On
OUT TR0
AND 1238.05  ; 后上料伺服到仓3放料位置(A)
AND>SL(323) D3300 D3340  ; 后腔体上料伺服当前位置, 腔体3检测有料开始位置
AND<SL(313) D3300 D3342  ; 后腔体上料伺服当前位置, 腔体3检测最后位置
AND 0.07  ; 后腔体有料感应
OUT TR1
AND T1318  ; 腔体3判断有料延时
SET H23.08  ; 腔体3有料
LD TR1
TIMHX(551) 1318 &4  ; 腔体3判断有料延时
LD TR0
AND 1238.06  ; 后上料伺服到仓4放料位置(A)
AND>SL(323) D3300 D3344  ; 后腔体上料伺服当前位置, 腔体4检测有料开始位置
AND<SL(313) D3300 D3346  ; 后腔体上料伺服当前位置, 腔体4检测最后位置
AND 0.07  ; 后腔体有料感应
OUT TR0
AND T1319  ; 腔体4判断有料延时
SET H24.08  ; 腔体4有料
LD TR0
TIMHX(551) 1319 &4  ; 腔体4判断有料延时
; rung 16: 定位到指定位置
LDNOT A326.05  ; 后上料伺服无原点标志
OUT TR0
AND T0238  ; 后腔体进料机械手升降气缸缩回位
AND 2962.06  ; 后腔体上料伺服正转极限
AND 2962.07  ; 后腔体上料伺服反转极限
ANDNOT A326.04  ; 后上料伺服脉冲输出中
AND T0320  ; 后上料伺服Ready
ANDNOT T0321  ; 后上料伺服报警
OUT 1238.11  ; 后上料伺服自动定位条件
LD TR0
AND 1238.12  ; 后上料伺服自动定位(A)
ANDNOT A326.04  ; 后上料伺服脉冲输出中
AND 100.05  ; 停止中
@PLS2(887) #2 #101 D2320 D2326  ; 后上料伺服自动加速比率, 后上料伺服自动启动速度
; rung 17
ILC(003)
; rung 18
LD T0000  ; PLC上电
AND 37.05  ; 后上料夹爪气缸松开按钮
RSET H53.00  ; 后上料夹爪有料
RSET H11.03  ; 后上料夹爪夹紧

### Section 外部输出

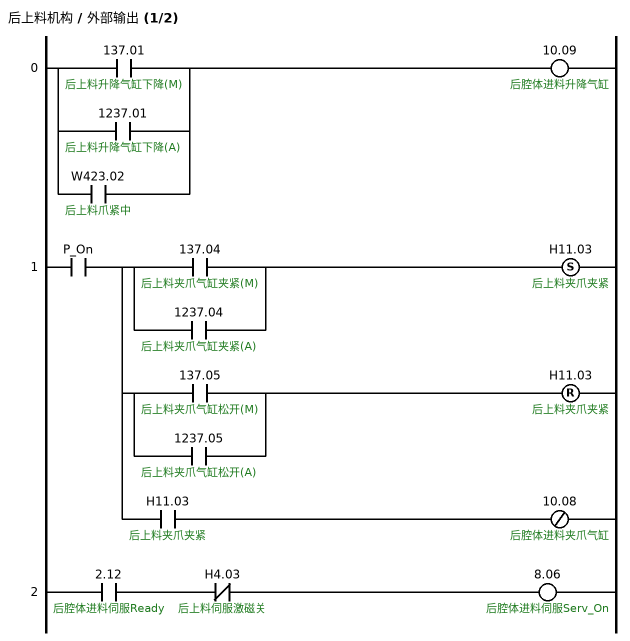
; rung 0
LD 137.01  ; 后上料升降气缸下降(M)
OR 1237.01  ; 后上料升降气缸下降(A)
OR W423.02  ; 后上料爪紧中
OUT 10.09  ; 后腔体进料升降气缸
; rung 1
LD P_On
OUT TR0
LD 137.04  ; 后上料夹爪气缸夹紧(M)
OR 1237.04  ; 后上料夹爪气缸夹紧(A)
ANDLD
SET H11.03  ; 后上料夹爪夹紧
LD TR0
LD 137.05  ; 后上料夹爪气缸松开(M)
OR 1237.05  ; 后上料夹爪气缸松开(A)
ANDLD
RSET H11.03  ; 后上料夹爪夹紧
LD TR0
AND H11.03  ; 后上料夹爪夹紧
OUTNOT 10.08  ; 后腔体进料夹爪气缸
; rung 2
LD 2.12  ; 后腔体进料伺服Ready
ANDNOT H4.03  ; 后上料伺服激磁关
OUT 8.06  ; 后腔体进料伺服Serv_On

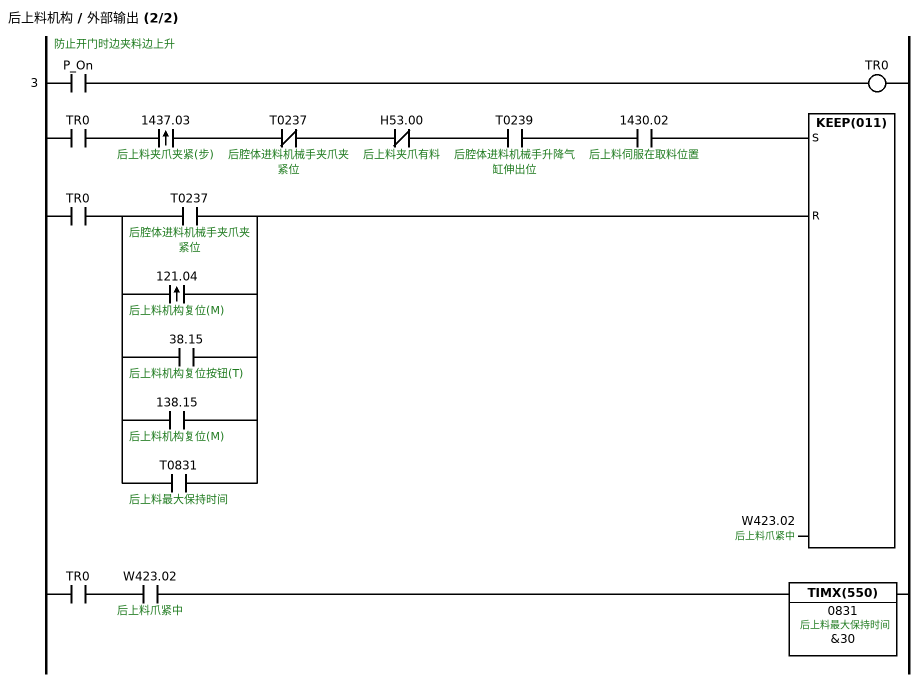
; rung 3: 防止开门时边夹料边上升
LD P_On
OUT TR0
@AND 1437.03  ; 后上料夹爪夹紧(步)
ANDNOT T0237  ; 后腔体进料机械手夹爪夹紧位
ANDNOT H53.00  ; 后上料夹爪有料
AND T0239  ; 后腔体进料机械手升降气缸伸出位
AND 1430.02  ; 后上料伺服在取料位置
LD TR0
LD T0237  ; 后腔体进料机械手夹爪夹紧位
@OR 121.04  ; 后上料机构复位(M)
OR 38.15  ; 后上料机构复位按钮(T)
OR 138.15  ; 后上料机构复位(M)
OR T0831  ; 后上料最大保持时间
ANDLD
KEEP(011) W423.02  ; 后上料爪紧中
LD TR0
AND W423.02  ; 后上料爪紧中
TIMX(550) 0831 &30  ; 后上料最大保持时间

### Section 指示灯
; rung 0: ************************************************** / 气缸动作及位置指示灯

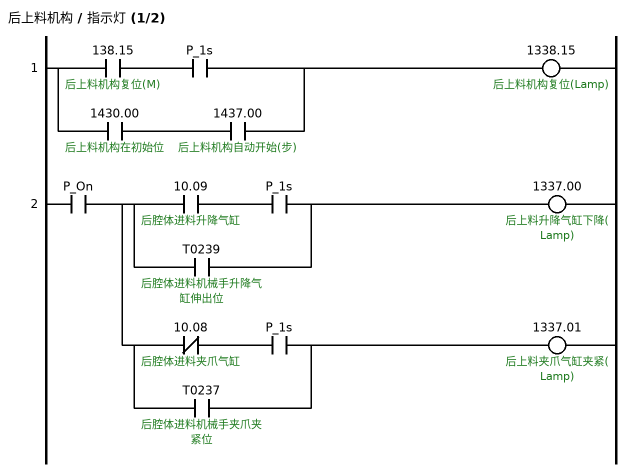
; rung 1
LD 138.15  ; 后上料机构复位(M)
AND P_1s
LD 1430.00  ; 后上料机构在初始位
AND 1437.00  ; 后上料机构自动开始(步)
ORLD
OUT 1338.15  ; 后上料机构复位(Lamp)
; rung 2
LD P_On
OUT TR0
LD 10.09  ; 后腔体进料升降气缸
AND P_1s
OR T0239  ; 后腔体进料机械手升降气缸伸出位
ANDLD
OUT 1337.00  ; 后上料升降气缸下降(Lamp)
LD TR0
LDNOT 10.08  ; 后腔体进料夹爪气缸
AND P_1s
OR T0237  ; 后腔体进料机械手夹爪夹紧位
ANDLD
OUT 1337.01  ; 后上料夹爪气缸夹紧(Lamp)

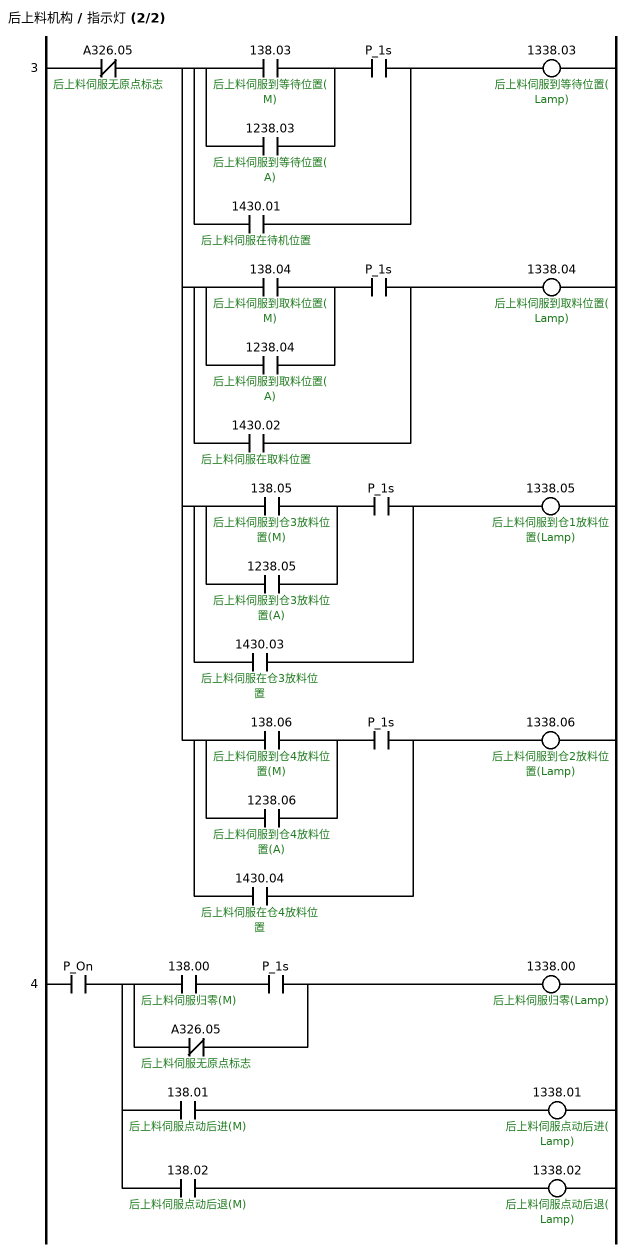
; rung 3
LDNOT A326.05  ; 后上料伺服无原点标志
OUT TR0
LD 138.03  ; 后上料伺服到等待位置(M)
OR 1238.03  ; 后上料伺服到等待位置(A)
AND P_1s
OR 1430.01  ; 后上料伺服在待机位置
ANDLD
OUT 1338.03  ; 后上料伺服到等待位置(Lamp)
LD TR0
LD 138.04  ; 后上料伺服到取料位置(M)
OR 1238.04  ; 后上料伺服到取料位置(A)
AND P_1s
OR 1430.02  ; 后上料伺服在取料位置
ANDLD
OUT 1338.04  ; 后上料伺服到取料位置(Lamp)
LD TR0
LD 138.05  ; 后上料伺服到仓3放料位置(M)
OR 1238.05  ; 后上料伺服到仓3放料位置(A)
AND P_1s
OR 1430.03  ; 后上料伺服在仓3放料位置
ANDLD
OUT 1338.05  ; 后上料伺服到仓1放料位置(Lamp)
LD TR0
LD 138.06  ; 后上料伺服到仓4放料位置(M)
OR 1238.06  ; 后上料伺服到仓4放料位置(A)
AND P_1s
OR 1430.04  ; 后上料伺服在仓4放料位置
ANDLD
OUT 1338.06  ; 后上料伺服到仓2放料位置(Lamp)
; rung 4
LD P_On
OUT TR0
LD 138.00  ; 后上料伺服归零(M)
AND P_1s
ORNOT A326.05  ; 后上料伺服无原点标志
ANDLD
OUT 1338.00  ; 后上料伺服归零(Lamp)
LD TR0
AND 138.01  ; 后上料伺服点动后进(M)
OUT 1338.01  ; 后上料伺服点动后进(Lamp)
LD TR0
AND 138.02  ; 后上料伺服点动后退(M)
OUT 1338.02  ; 后上料伺服点动后退(Lamp)

### Section END
; rung 0
END(001)

## Program 后下料机构 (cyclic task 5)

### Section Main

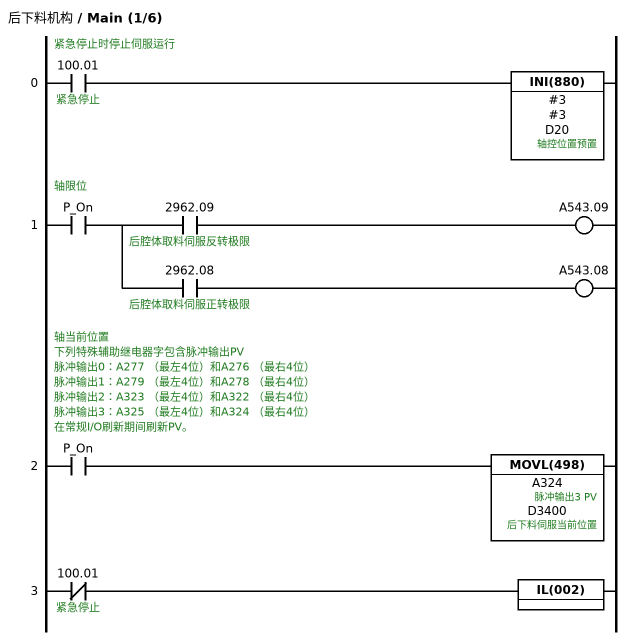
; rung 0: 紧急停止时停止伺服运行
LD 100.01  ; 紧急停止
INI(880) #3 #3 D20  ; 轴控位置预置
; rung 1: 轴限位
LD P_On
OUT TR0
AND 2962.09  ; 后腔体取料伺服反转极限
OUT A543.09
LD TR0
AND 2962.08  ; 后腔体取料伺服正转极限
OUT A543.08
; rung 2: 轴当前位置 / 下列特殊辅助继电器字包含脉冲输出PV / 脉冲输出0：A277 （最左4位）和A276 （最右4位） / 脉冲输出1：A279 （最左4位）和A278 （最右4位） / 脉冲输出2：A323 （最左4位）和A322 （最右4位） / 脉冲输出3：A325 （最左4位）和A324 （最右4位） / 在常规I/O刷新期间刷新PV。
LD P_On
MOVL(498) A324 D3400  ; 脉冲输出3 PV, 后下料伺服当前位置
; rung 3
LDNOT 100.01  ; 紧急停止
IL(002)

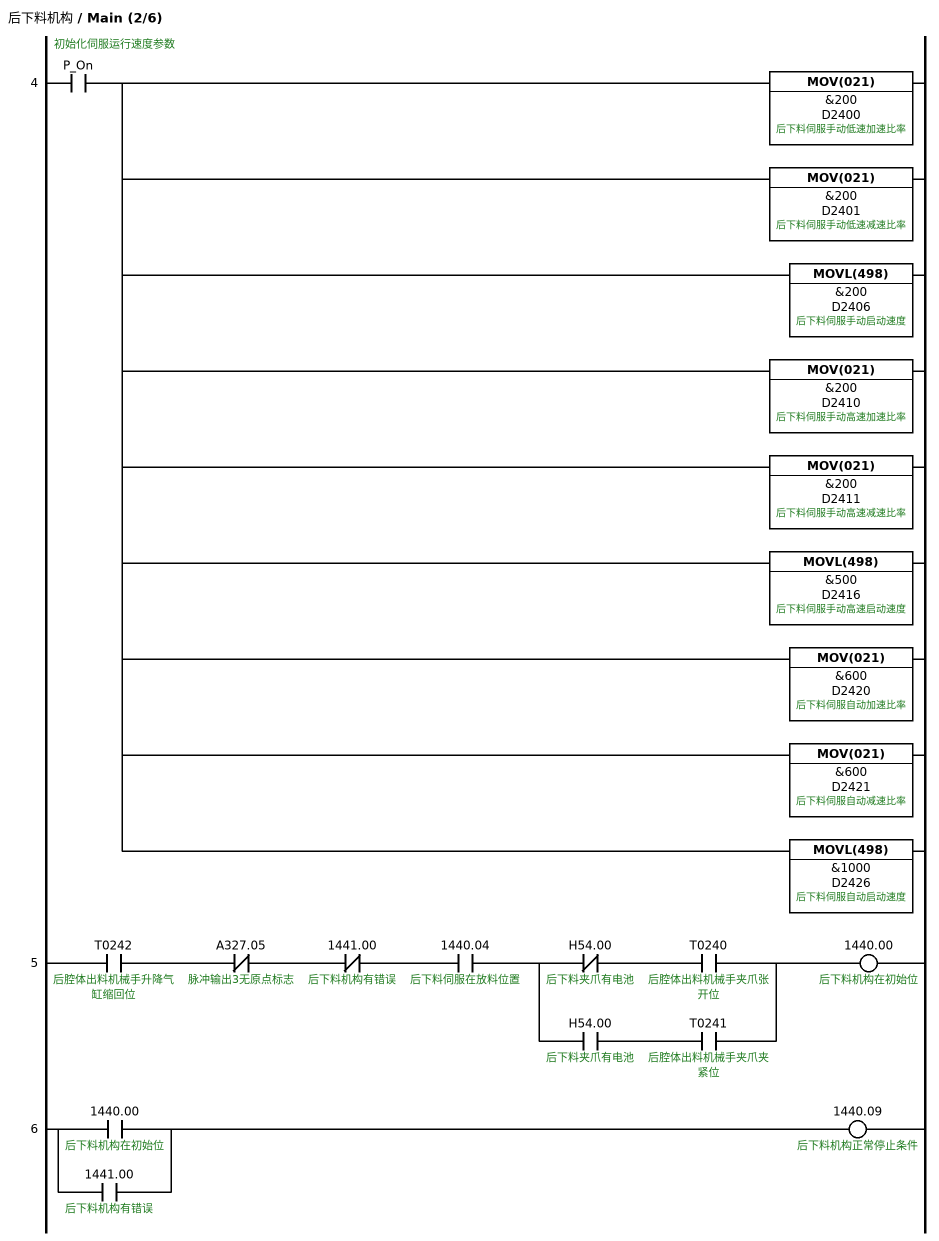
; rung 4: 初始化伺服运行速度参数
LD P_On
MOV(021) &200 D2400  ; 后下料伺服手动低速加速比率
MOV(021) &200 D2401  ; 后下料伺服手动低速减速比率
MOVL(498) &200 D2406  ; 后下料伺服手动启动速度
MOV(021) &200 D2410  ; 后下料伺服手动高速加速比率
MOV(021) &200 D2411  ; 后下料伺服手动高速减速比率
MOVL(498) &500 D2416  ; 后下料伺服手动高速启动速度
MOV(021) &600 D2420  ; 后下料伺服自动加速比率
MOV(021) &600 D2421  ; 后下料伺服自动减速比率
MOVL(498) &1000 D2426  ; 后下料伺服自动启动速度
; rung 5
LD T0242  ; 后腔体出料机械手升降气缸缩回位
ANDNOT A327.05  ; 脉冲输出3无原点标志
ANDNOT 1441.00  ; 后下料机构有错误
AND 1440.04  ; 后下料伺服在放料位置
LDNOT H54.00  ; 后下料夹爪有电池
AND T0240  ; 后腔体出料机械手夹爪张开位
LD H54.00  ; 后下料夹爪有电池
AND T0241  ; 后腔体出料机械手夹爪夹紧位
ORLD
ANDLD
OUT 1440.00  ; 后下料机构在初始位
; rung 6
LD 1440.00  ; 后下料机构在初始位
OR 1441.00  ; 后下料机构有错误
OUT 1440.09  ; 后下料机构正常停止条件

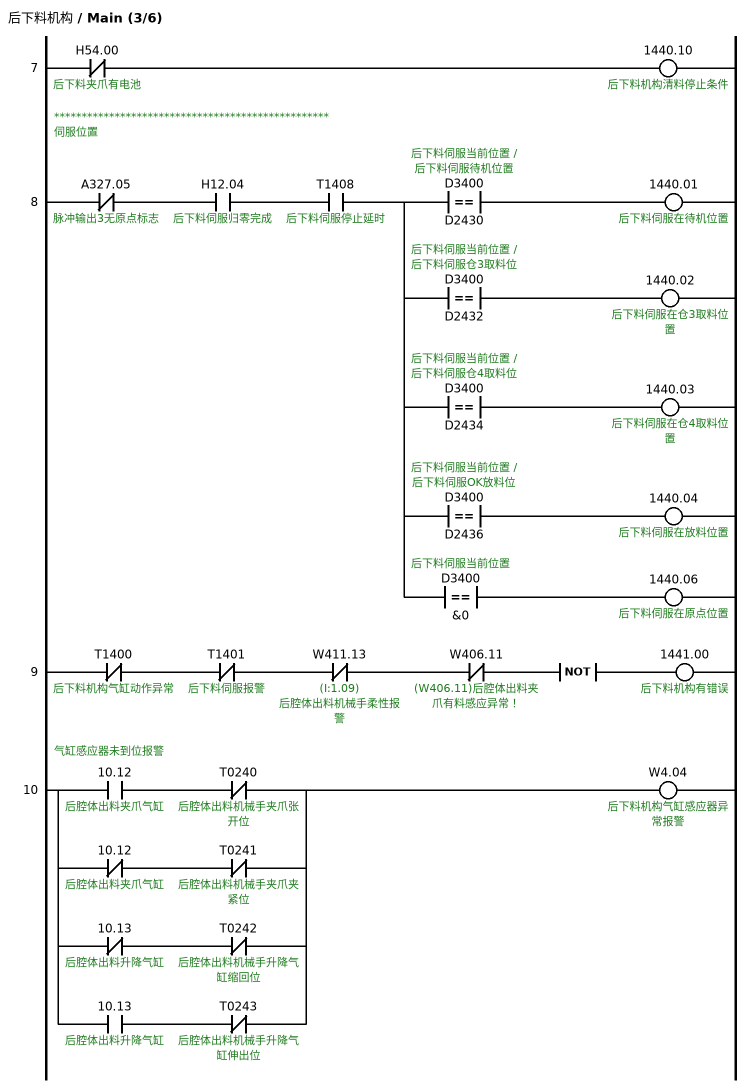
; rung 7
LDNOT H54.00  ; 后下料夹爪有电池
OUT 1440.10  ; 后下料机构清料停止条件
; rung 8: ************************************************** / 伺服位置
LDNOT A327.05  ; 脉冲输出3无原点标志
AND H12.04  ; 后下料伺服归零完成
AND T1408  ; 后下料伺服停止延时
OUT TR0
AND=SL(303) D3400 D2430  ; 后下料伺服当前位置, 后下料伺服待机位置
OUT 1440.01  ; 后下料伺服在待机位置
LD TR0
AND=SL(303) D3400 D2432  ; 后下料伺服当前位置, 后下料伺服仓3取料位
OUT 1440.02  ; 后下料伺服在仓3取料位置
LD TR0
AND=SL(303) D3400 D2434  ; 后下料伺服当前位置, 后下料伺服仓4取料位
OUT 1440.03  ; 后下料伺服在仓4取料位置
LD TR0
AND=SL(303) D3400 D2436  ; 后下料伺服当前位置, 后下料伺服OK放料位
OUT 1440.04  ; 后下料伺服在放料位置
LD TR0
AND=SL(303) D3400 &0  ; 后下料伺服当前位置
OUT 1440.06  ; 后下料伺服在原点位置
; rung 9
LDNOT T1400  ; 后下料机构气缸动作异常
ANDNOT T1401  ; 后下料伺服报警
ANDNOT W411.13  ; (I:1.09) 后腔体出料机械手柔性报警
ANDNOT W406.11  ; (W406.11)后腔体出料夹爪有料感应异常！
NOT(520)
OUT 1441.00  ; 后下料机构有错误
; rung 10: 气缸感应器未到位报警
LD 10.12  ; 后腔体出料夹爪气缸
ANDNOT T0240  ; 后腔体出料机械手夹爪张开位
LDNOT 10.12  ; 后腔体出料夹爪气缸
ANDNOT T0241  ; 后腔体出料机械手夹爪夹紧位
ORLD
LDNOT 10.13  ; 后腔体出料升降气缸
ANDNOT T0242  ; 后腔体出料机械手升降气缸缩回位
ORLD
LD 10.13  ; 后腔体出料升降气缸
ANDNOT T0243  ; 后腔体出料机械手升降气缸伸出位
ORLD
OUT W4.04  ; 后下料机构气缸感应器异常报警

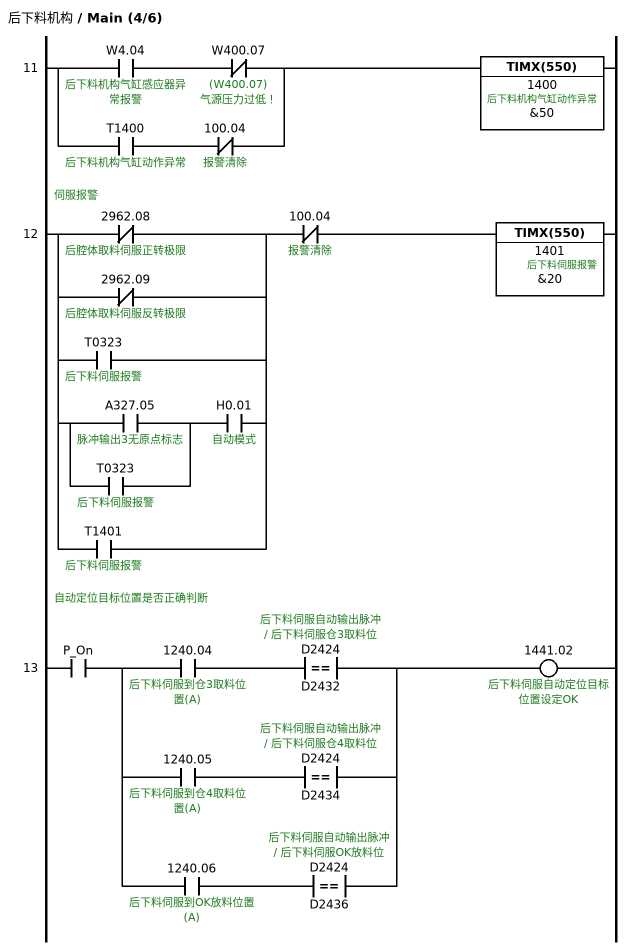
; rung 11
LD W4.04  ; 后下料机构气缸感应器异常报警
ANDNOT W400.07  ; (W400.07) 气源压力过低！
LD T1400  ; 后下料机构气缸动作异常
ANDNOT 100.04  ; 报警清除
ORLD
TIMX(550) 1400 &50  ; 后下料机构气缸动作异常
; rung 12: 伺服报警
LDNOT 2962.08  ; 后腔体取料伺服正转极限
ORNOT 2962.09  ; 后腔体取料伺服反转极限
OR T0323  ; 后下料伺服报警
LD A327.05  ; 脉冲输出3无原点标志
OR T0323  ; 后下料伺服报警
AND H0.01  ; 自动模式
ORLD
OR T1401  ; 后下料伺服报警
ANDNOT 100.04  ; 报警清除
TIMX(550) 1401 &20  ; 后下料伺服报警
; rung 13: 自动定位目标位置是否正确判断
LD P_On
LD 1240.04  ; 后下料伺服到仓3取料位置(A)
AND=SL(303) D2424 D2432  ; 后下料伺服自动输出脉冲, 后下料伺服仓3取料位
LD 1240.05  ; 后下料伺服到仓4取料位置(A)
AND=SL(303) D2424 D2434  ; 后下料伺服自动输出脉冲, 后下料伺服仓4取料位
ORLD
LD 1240.06  ; 后下料伺服到OK放料位置(A)
AND=SL(303) D2424 D2436  ; 后下料伺服自动输出脉冲, 后下料伺服OK放料位
ORLD
ANDLD
OUT 1441.02  ; 后下料伺服自动定位目标位置设定OK

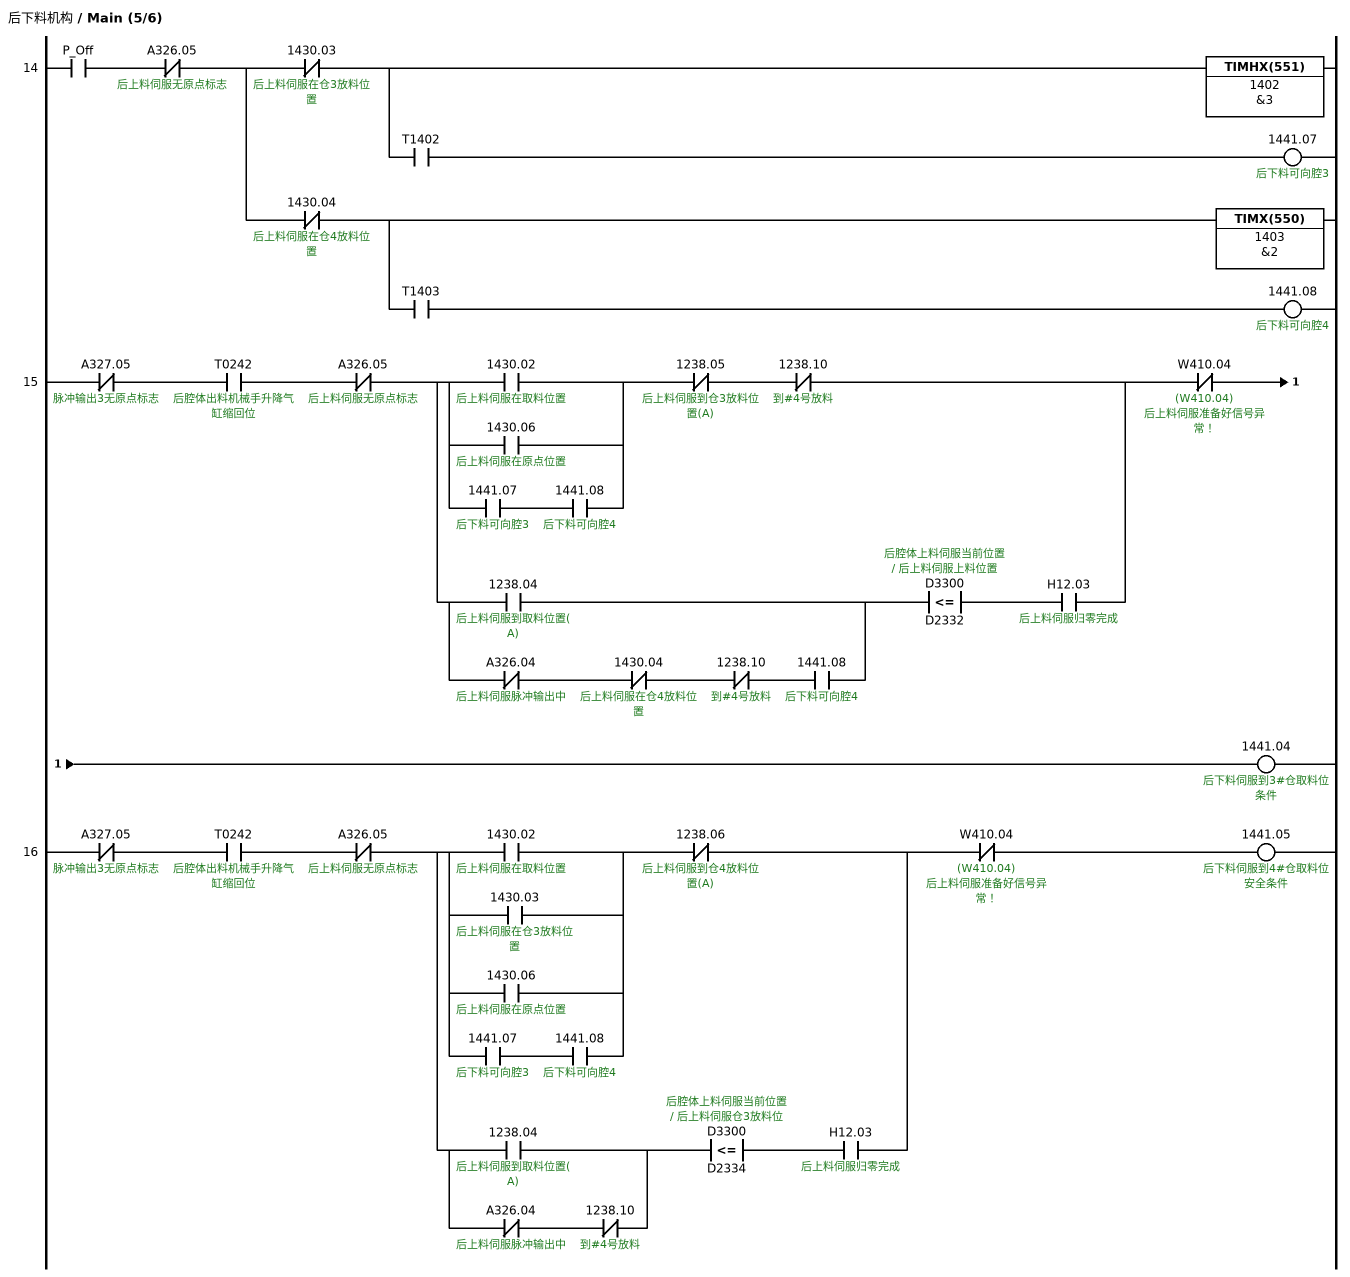
; rung 14
LD P_Off
ANDNOT A326.05  ; 后上料伺服无原点标志
OUT TR0
ANDNOT 1430.03  ; 后上料伺服在仓3放料位置
TIMHX(551) 1402 &3
AND T1402
OUT 1441.07  ; 后下料可向腔3
LD TR0
ANDNOT 1430.04  ; 后上料伺服在仓4放料位置
TIMX(550) 1403 &2
AND T1403
OUT 1441.08  ; 后下料可向腔4
; rung 15
LDNOT A327.05  ; 脉冲输出3无原点标志
AND T0242  ; 后腔体出料机械手升降气缸缩回位
ANDNOT A326.05  ; 后上料伺服无原点标志
LD 1430.02  ; 后上料伺服在取料位置
OR 1430.06  ; 后上料伺服在原点位置
LD 1441.07  ; 后下料可向腔3
AND 1441.08  ; 后下料可向腔4
ORLD
ANDNOT 1238.05  ; 后上料伺服到仓3放料位置(A)
ANDNOT 1238.10  ; 到#4号放料
LD 1238.04  ; 后上料伺服到取料位置(A)
LDNOT A326.04  ; 后上料伺服脉冲输出中
ANDNOT 1430.04  ; 后上料伺服在仓4放料位置
ANDNOT 1238.10  ; 到#4号放料
AND 1441.08  ; 后下料可向腔4
ORLD
AND<=SL(318) D3300 D2332  ; 后腔体上料伺服当前位置, 后上料伺服上料位置
AND H12.03  ; 后上料伺服归零完成
ORLD
ANDLD
ANDNOT W410.04  ; (W410.04) 后上料伺服准备好信号异常！
OUT 1441.04  ; 后下料伺服到3#仓取料位条件
; rung 16
LDNOT A327.05  ; 脉冲输出3无原点标志
AND T0242  ; 后腔体出料机械手升降气缸缩回位
ANDNOT A326.05  ; 后上料伺服无原点标志
LD 1430.02  ; 后上料伺服在取料位置
OR 1430.03  ; 后上料伺服在仓3放料位置
OR 1430.06  ; 后上料伺服在原点位置
LD 1441.07  ; 后下料可向腔3
AND 1441.08  ; 后下料可向腔4
ORLD
ANDNOT 1238.06  ; 后上料伺服到仓4放料位置(A)
LD 1238.04  ; 后上料伺服到取料位置(A)
LDNOT A326.04  ; 后上料伺服脉冲输出中
ANDNOT 1238.10  ; 到#4号放料
ORLD
AND<=SL(318) D3300 D2334  ; 后腔体上料伺服当前位置, 后上料伺服仓3放料位
AND H12.03  ; 后上料伺服归零完成
ORLD
ANDLD
ANDNOT W410.04  ; (W410.04) 后上料伺服准备好信号异常！
OUT 1441.05  ; 后下料伺服到4#仓取料位安全条件

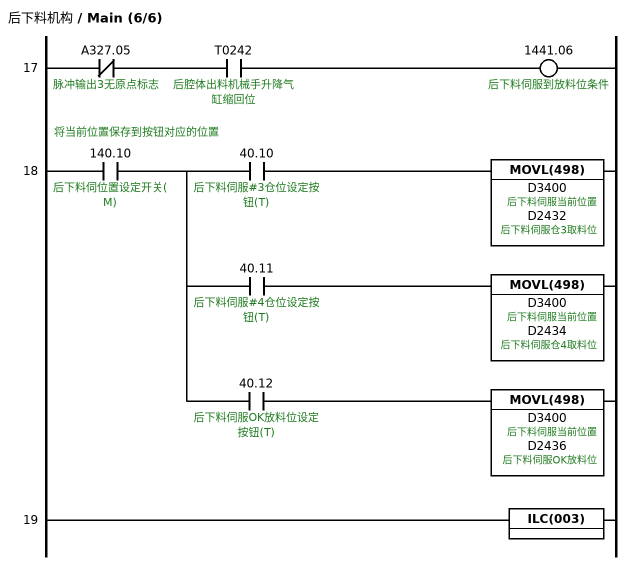
; rung 17
LDNOT A327.05  ; 脉冲输出3无原点标志
AND T0242  ; 后腔体出料机械手升降气缸缩回位
OUT 1441.06  ; 后下料伺服到放料位条件
; rung 18: 将当前位置保存到按钮对应的位置
LD 140.10  ; 后下料伺位置设定开关(M)
OUT TR0
AND 40.10  ; 后下料伺服#3仓位设定按钮(T)
MOVL(498) D3400 D2432  ; 后下料伺服当前位置, 后下料伺服仓3取料位
LD TR0
AND 40.11  ; 后下料伺服#4仓位设定按钮(T)
MOVL(498) D3400 D2434  ; 后下料伺服当前位置, 后下料伺服仓4取料位
LD TR0
AND 40.12  ; 后下料伺服OK放料位设定按钮(T)
MOVL(498) D3400 D2436  ; 后下料伺服当前位置, 后下料伺服OK放料位
; rung 19
ILC(003)

### Section 工站复位

